C05458=1026.978,-87.134,412.335,166.934,44.993,158.253
C05459=1026.984,-86.885,412.325,166.937,44.991,158.253
C05460=1026.990,-86.635,412.315,166.940,44.988,158.253
C05461=1026.996,-86.385,412.304,166.943,44.986,158.253
C05462=1027.001,-86.135,412.294,166.946,44.984,158.253
C05463=1027.008,-85.886,412.284,166.948,44.981,158.252
C05464=1027.013,-85.636,412.274,166.952,44.979,158.252
C05465=1027.019,-85.386,412.264,166.954,44.976,158.252
C05466=1027.026,-85.103,412.252,166.958,44.974,158.252
C05467=1027.033,-84.819,412.240,166.961,44.971,158.252
C05468=1027.040,-84.534,412.228,166.965,44.968,158.252
C05469=1027.046,-84.250,412.217,166.968,44.966,158.252
C05470=1027.053,-84.001,412.207,166.971,44.964,158.251
C05471=1027.058,-83.751,412.196,166.974,44.961,158.251
C05472=1027.065,-83.502,412.186,166.977,44.959,158.251
C05473=1027.070,-83.252,412.176,166.980,44.956,158.251
C05474=1027.077,-83.002,412.165,166.983,44.954,158.251
C05475=1027.083,-82.752,412.155,166.986,44.952,158.251
C05476=1027.088,-82.502,412.144,166.989,44.949,158.251
C05477=1027.094,-82.252,412.135,166.992,44.947,158.251
C05478=1027.100,-82.003,412.124,166.995,44.944,158.250
C05479=1027.107,-81.754,412.114,166.997,44.942,158.250
C05480=1027.112,-81.503,412.103,167.001,44.939,158.250
C05481=1027.119,-81.254,412.093,167.003,44.937,158.250
C05482=1027.125,-81.003,412.083,167.007,44.934,158.250
C05483=1027.130,-80.754,412.072,167.009,44.932,158.250
C05484=1027.137,-80.505,412.061,167.013,44.929,158.250
C05485=1027.142,-80.255,412.051,167.015,44.927,158.250
C05486=1027.149,-80.006,412.041,167.019,44.925,158.250
C05487=1027.154,-79.756,412.030,167.021,44.922,158.249
C05488=1027.161,-79.505,412.020,167.024,44.920,158.249
C05489=1027.166,-79.256,412.009,167.027,44.918,158.249
C05490=1027.172,-79.006,411.998,167.030,44.916,158.249
C05491=1027.178,-78.757,411.988,167.032,44.914,158.249
C05492=1027.184,-78.507,411.977,167.036,44.911,158.249
C05493=1027.190,-78.257,411.966,167.038,44.909,158.249
C05494=1027.196,-78.007,411.955,167.042,44.907,158.249
C05495=1027.202,-77.758,411.944,167.044,44.905,158.248
C05496=1027.207,-77.508,411.934,167.047,44.903,158.248
C05497=1027.214,-77.258,411.924,167.050,44.900,158.248
C05498=1027.220,-77.008,411.913,167.053,44.898,158.248
C05499=1027.226,-76.759,411.902,167.056,44.896,158.248
C05500=1027.231,-76.509,411.891,167.059,44.893,158.248
C05501=1027.237,-76.260,411.880,167.062,44.891,158.248
C05502=1027.243,-76.010,411.869,167.065,44.889,158.248
C05503=1027.250,-75.760,411.859,167.068,44.887,158.248
C05504=1027.255,-75.510,411.848,167.070,44.884,158.247
C05505=1027.261,-75.261,411.838,167.074,44.882,158.247
C05506=1027.267,-75.011,411.827,167.076,44.880,158.247
C05507=1027.273,-74.761,411.815,167.079,44.877,158.247
C05508=1027.279,-74.512,411.805,167.082,44.875,158.247
C05509=1027.285,-74.262,411.794,167.085,44.873,158.247
C05510=1027.290,-74.013,411.783,167.089,44.871,158.247
C05511=1027.297,-73.763,411.772,167.091,44.868,158.247
C05512=1027.303,-73.513,411.761,167.094,44.866,158.247
C05513=1027.308,-73.264,411.750,167.096,44.864,158.246
C05514=1027.315,-73.013,411.739,167.100,44.862,158.246
C05515=1027.320,-72.764,411.728,167.102,44.860,158.246
C05516=1027.326,-72.514,411.717,167.105,44.858,158.246
C05517=1027.331,-72.265,411.705,167.109,44.856,158.246
C05518=1027.337,-72.014,411.694,167.111,44.854,158.246
C05519=1027.343,-71.765,411.683,167.113,44.851,158.246
C05520=1027.349,-71.515,411.672,167.117,44.849,158.246
C05521=1027.355,-71.265,411.661,167.120,44.847,158.246
C05522=1027.361,-71.016,411.650,167.122,44.845,158.246
C05523=1027.367,-70.766,411.639,167.125,44.843,158.246
C05524=1027.373,-70.517,411.627,167.129,44.841,158.246
C05525=1027.378,-70.267,411.616,167.131,44.839,158.245
C05526=1027.384,-70.017,411.605,167.134,44.837,158.245
C05527=1027.390,-69.767,411.594,167.137,44.834,158.245
C05528=1027.396,-69.518,411.583,167.140,44.832,158.245
C05529=1027.402,-69.268,411.572,167.142,44.830,158.245
C05530=1027.408,-68.987,411.559,167.146,44.828,158.245
C05531=1027.416,-68.704,411.546,167.149,44.825,158.245
C05532=1027.422,-68.423,411.534,167.152,44.823,158.245
C05533=1027.428,-68.141,411.521,167.155,44.820,158.245
C05534=1027.435,-67.891,411.509,167.158,44.818,158.244
C05535=1027.441,-67.641,411.498,167.161,44.816,158.244
C05536=1027.447,-67.391,411.487,167.164,44.814,158.244
C05537=1027.453,-67.142,411.476,167.167,44.812,158.244
C05538=1027.458,-66.892,411.465,167.170,44.810,158.244
C05539=1027.464,-66.642,411.453,167.173,44.807,158.244
C05540=1027.470,-66.393,411.442,167.175,44.805,158.244
C05541=1027.476,-66.143,411.430,167.178,44.803,158.244
C05542=1027.482,-65.894,411.419,167.181,44.801,158.244
C05543=1027.488,-65.644,411.408,167.184,44.799,158.244
C05544=1027.494,-65.394,411.396,167.187,44.797,158.244
C05545=1027.499,-65.144,411.385,167.190,44.794,158.243
C05546=1027.506,-64.895,411.373,167.193,44.792,158.243
C05547=1027.512,-64.645,411.362,167.195,44.790,158.243
C05548=1027.518,-64.395,411.351,167.199,44.788,158.243
C05549=1027.524,-64.146,411.340,167.201,44.786,158.243
C05550=1027.530,-63.896,411.328,167.204,44.784,158.243
C05551=1027.536,-63.646,411.317,167.206,44.781,158.243
C05552=1027.542,-63.397,411.305,167.210,44.779,158.243
C05553=1027.548,-63.147,411.294,167.213,44.777,158.243
C05554=1027.555,-62.898,411.282,167.215,44.775,158.242
C05555=1027.560,-62.648,411.271,167.219,44.773,158.242
C05556=1027.566,-62.398,411.259,167.221,44.770,158.242
C05557=1027.572,-62.149,411.248,167.224,44.768,158.242
C05558=1027.578,-61.899,411.237,167.227,44.766,158.242
C05559=1027.584,-61.650,411.225,167.230,44.764,158.242
C05560=1027.590,-61.399,411.213,167.233,44.762,158.242
C05561=1027.596,-61.150,411.202,167.235,44.760,158.242
C05562=1027.602,-60.900,411.190,167.239,44.757,158.242
C05563=1027.608,-60.651,411.179,167.241,44.755,158.241
C05564=1027.615,-60.401,411.167,167.244,44.753,158.241
C05565=1027.620,-60.151,411.156,167.247,44.751,158.241
C05566=1027.626,-59.902,411.144,167.250,44.749,158.241
C05567=1027.633,-59.652,411.133,167.252,44.747,158.241
C05568=1027.639,-59.403,411.121,167.255,44.745,158.241
C05569=1027.645,-59.152,411.110,167.259,44.742,158.241
C05570=1027.650,-58.903,411.098,167.261,44.740,158.241
C05571=1027.657,-58.653,411.086,167.264,44.738,158.241
C05572=1027.663,-58.404,411.075,167.267,44.736,158.240
C05573=1027.669,-58.154,411.064,167.270,44.734,158.240
C05574=1027.676,-57.904,411.052,167.272,44.732,158.240
C05575=1027.681,-57.655,411.040,167.276,44.729,158.240
C05576=1027.687,-57.405,411.028,167.278,44.727,158.240
C05577=1027.694,-57.155,411.017,167.281,44.725,158.240
C05578=1027.700,-56.906,411.005,167.284,44.723,158.240
C05579=1027.706,-56.656,410.993,167.287,44.721,158.240
C05580=1027.712,-56.407,410.982,167.289,44.718,158.240
C05581=1027.718,-56.157,410.970,167.292,44.716,158.239
C05582=1027.725,-55.907,410.959,167.296,44.714,158.239
C05583=1027.731,-55.658,410.947,167.298,44.712,158.239
C05584=1027.736,-55.408,410.935,167.301,44.709,158.239
C05585=1027.743,-55.158,410.923,167.303,44.707,158.239
C05586=1027.749,-54.909,410.912,167.307,44.705,158.239
C05587=1027.756,-54.660,410.900,167.309,44.703,158.239
C05588=1027.761,-54.409,410.888,167.312,44.700,158.239
C05589=1027.768,-54.159,410.876,167.315,44.698,158.239
C05590=1027.774,-53.911,410.864,167.318,44.696,158.238
C05591=1027.780,-53.660,410.853,167.321,44.694,158.238
C05592=1027.786,-53.410,410.841,167.324,44.692,158.238
C05593=1027.792,-53.162,410.829,167.327,44.690,158.238
C05594=1027.799,-52.881,410.816,167.329,44.687,158.238
C05595=1027.806,-52.600,410.802,167.333,44.685,158.238
C05596=1027.813,-52.319,410.790,167.336,44.682,158.238
C05597=1027.821,-52.038,410.776,167.340,44.680,158.238
C05598=1027.826,-51.788,410.764,167.342,44.678,158.237
C05599=1027.832,-51.539,410.753,167.345,44.675,158.237
C05600=1027.839,-51.290,410.741,167.347,44.673,158.237
C05601=1027.846,-51.040,410.729,167.351,44.671,158.237
C05602=1027.851,-50.789,410.717,167.353,44.668,158.237
C05603=1027.858,-50.540,410.705,167.356,44.666,158.237
C05604=1027.863,-50.291,410.693,167.358,44.664,158.237
C05605=1027.869,-50.041,410.680,167.362,44.662,158.237
C05606=1027.876,-49.791,410.668,167.365,44.660,158.236
C05607=1027.882,-49.541,410.656,167.367,44.658,158.236
C05608=1027.888,-49.293,410.644,167.370,44.656,158.236
C05609=1027.894,-49.043,410.631,167.372,44.654,158.236
C05610=1027.900,-48.793,410.619,167.376,44.652,158.236
C05611=1027.906,-48.543,410.607,167.379,44.650,158.236
C05612=1027.912,-48.294,410.595,167.381,44.648,158.236
C05613=1027.917,-48.044,410.582,167.384,44.646,158.236
C05614=1027.924,-47.795,410.570,167.386,44.644,158.236
C05615=1027.930,-47.545,410.558,167.389,44.642,158.236
C05616=1027.937,-47.295,410.546,167.393,44.640,158.236
C05617=1027.942,-47.046,410.534,167.395,44.638,158.235
C05618=1027.948,-46.796,410.521,167.398,44.636,158.235
C05619=1027.954,-46.546,410.509,167.400,44.634,158.235
C05620=1027.960,-46.297,410.497,167.403,44.632,158.235
C05621=1027.966,-46.047,410.484,167.407,44.630,158.235
C05622=1027.972,-45.798,410.472,167.409,44.628,158.235
C05623=1027.978,-45.548,410.460,167.412,44.626,158.235
C05624=1027.984,-45.298,410.447,167.414,44.624,158.235
C05625=1027.991,-45.048,410.435,167.417,44.622,158.235
C05626=1027.997,-44.799,410.423,167.420,44.619,158.235
C05627=1028.003,-44.549,410.410,167.423,44.617,158.234
C05628=1028.009,-44.300,410.399,167.426,44.615,158.234
C05629=1028.015,-44.050,410.386,167.428,44.614,158.234
C05630=1028.020,-43.800,410.373,167.431,44.612,158.234
C05631=1028.027,-43.551,410.361,167.433,44.610,158.234
C05632=1028.033,-43.301,410.348,167.437,44.607,158.234
C05633=1028.039,-43.051,410.336,167.440,44.605,158.234
C05634=1028.046,-42.802,410.324,167.442,44.604,158.234
C05635=1028.052,-42.552,410.311,167.445,44.602,158.234
C05636=1028.058,-42.302,410.299,167.447,44.600,158.234
C05637=1028.064,-42.052,410.287,167.451,44.597,158.233
C05638=1028.070,-41.804,410.274,167.453,44.595,158.233
C05639=1028.076,-41.554,410.261,167.456,44.593,158.233
C05640=1028.083,-41.304,410.249,167.459,44.591,158.233
C05641=1028.088,-41.055,410.237,167.461,44.589,158.233
C05642=1028.094,-40.805,410.224,167.464,44.587,158.233
C05643=1028.101,-40.556,410.211,167.467,44.585,158.233
C05644=1028.107,-40.306,410.199,167.470,44.583,158.233
C05645=1028.113,-40.056,410.186,167.473,44.581,158.233
C05646=1028.120,-39.806,410.174,167.475,44.579,158.232
C05647=1028.126,-39.557,410.161,167.478,44.576,158.232
C05648=1028.132,-39.307,410.149,167.481,44.574,158.232
C05649=1028.139,-39.058,410.137,167.484,44.572,158.232
C05650=1028.144,-38.808,410.124,167.486,44.570,158.232
C05651=1028.151,-38.558,410.111,167.489,44.568,158.232
C05652=1028.157,-38.309,410.098,167.492,44.566,158.232
C05653=1028.162,-38.059,410.086,167.494,44.564,158.232
C05654=1028.169,-37.809,410.072,167.497,44.562,158.232
C05655=1028.175,-37.560,410.060,167.499,44.560,158.231
C05656=1028.181,-37.310,410.047,167.503,44.558,158.231
C05657=1028.187,-37.060,410.034,167.506,44.557,158.231
C05658=1028.194,-36.780,410.019,167.508,44.554,158.231
C05659=1028.200,-36.500,410.006,167.512,44.552,158.231
C05660=1028.207,-36.220,409.991,167.514,44.550,158.231
C05661=1028.214,-35.940,409.977,167.518,44.548,158.231
C05662=1028.220,-35.690,409.963,167.521,44.546,158.231
C05663=1028.226,-35.440,409.951,167.523,44.544,158.231
C05664=1028.232,-35.191,409.938,167.526,44.542,158.231
C05665=1028.238,-34.941,409.925,167.528,44.540,158.231
C05666=1028.244,-34.691,409.913,167.531,44.538,158.230
C05667=1028.250,-34.442,409.899,167.534,44.536,158.230
C05668=1028.257,-34.193,409.887,167.536,44.534,158.230
C05669=1028.263,-33.943,409.874,167.539,44.532,158.230
C05670=1028.269,-33.693,409.861,167.542,44.530,158.230
C05671=1028.276,-33.443,409.848,167.545,44.528,158.230
C05672=1028.282,-33.194,409.835,167.548,44.526,158.230
C05673=1028.288,-32.944,409.822,167.550,44.524,158.230
C05674=1028.294,-32.695,409.809,167.553,44.522,158.230
C05675=1028.300,-32.445,409.796,167.555,44.520,158.230
C05676=1028.306,-32.196,409.783,167.558,44.519,158.229
C05677=1028.312,-31.946,409.770,167.561,44.517,158.229
C05678=1028.318,-31.697,409.757,167.563,44.515,158.229
C05679=1028.324,-31.447,409.745,167.567,44.512,158.229
C05680=1028.330,-31.198,409.731,167.570,44.511,158.229
C05681=1028.337,-30.948,409.718,167.572,44.509,158.229
C05682=1028.343,-30.698,409.705,167.575,44.507,158.229
C05683=1028.349,-30.448,409.692,167.577,44.505,158.229
C05684=1028.356,-30.199,409.679,167.580,44.502,158.228
C05685=1028.361,-29.949,409.666,167.582,44.500,158.228
C05686=1028.368,-29.700,409.653,167.585,44.498,158.228
C05687=1028.374,-29.450,409.640,167.587,44.496,158.228
C05688=1028.380,-29.201,409.627,167.591,44.494,158.228
C05689=1028.387,-28.951,409.613,167.594,44.492,158.228
C05690=1028.393,-28.701,409.601,167.596,44.490,158.228
C05691=1028.399,-28.452,409.587,167.599,44.488,158.228
C05692=1028.405,-28.203,409.574,167.602,44.486,158.228
C05693=1028.411,-27.953,409.562,167.604,44.484,158.228
C05694=1028.418,-27.703,409.548,167.607,44.482,158.227
C05695=1028.424,-27.453,409.535,167.609,44.480,158.227
C05696=1028.430,-27.204,409.521,167.612,44.478,158.227
C05697=1028.436,-26.954,409.509,167.615,44.476,158.227
C05698=1028.442,-26.705,409.496,167.617,44.475,158.227
C05699=1028.448,-26.456,409.482,167.620,44.473,158.227
C05700=1028.455,-26.205,409.468,167.623,44.470,158.227
C05701=1028.461,-25.956,409.455,167.626,44.468,158.227
C05702=1028.467,-25.707,409.442,167.629,44.467,158.227
C05703=1028.473,-25.457,409.429,167.631,44.465,158.227
C05704=1028.478,-25.207,409.415,167.634,44.463,158.227
C05705=1028.485,-24.958,409.402,167.637,44.461,158.226
C05706=1028.491,-24.708,409.388,167.639,44.459,158.226
C05707=1028.498,-24.459,409.375,167.642,44.457,158.226
C05708=1028.503,-24.209,409.361,167.644,44.456,158.226
C05709=1028.509,-23.960,409.348,167.647,44.454,158.226
C05710=1028.516,-23.710,409.334,167.650,44.452,158.226
C05711=1028.522,-23.460,409.322,167.652,44.450,158.226
C05712=1028.527,-23.211,409.308,167.655,44.448,158.226
C05713=1028.534,-22.961,409.295,167.657,44.446,158.226
C05714=1028.540,-22.718,409.281,167.660,44.445,158.226
C05715=1028.546,-22.474,409.268,167.663,44.443,158.226
C05716=1028.552,-22.230,409.255,167.665,44.441,158.225
C05717=1028.558,-21.987,409.241,167.668,44.439,158.225
C05718=1028.564,-21.743,409.228,167.671,44.437,158.225
C05719=1028.570,-21.499,409.215,167.673,44.435,158.225
C05720=1028.576,-21.255,409.201,167.676,44.433,158.225
C05721=1028.582,-21.011,409.189,167.678,44.431,158.225
C05722=1028.590,-20.718,409.173,167.681,44.429,158.225
C05723=1028.597,-20.426,409.157,167.685,44.427,158.225
C05724=1028.605,-20.133,409.141,167.687,44.424,158.224
C05725=1028.611,-19.841,409.125,167.691,44.422,158.224
C05726=1028.618,-19.591,409.111,167.693,44.420,158.224
C05727=1028.624,-19.341,409.098,167.696,44.418,158.224
C05728=1028.630,-19.092,409.084,167.698,44.416,158.224
C05729=1028.637,-18.842,409.070,167.701,44.414,158.224
C05730=1028.643,-18.593,409.057,167.704,44.412,158.224
C05731=1028.648,-18.343,409.043,167.706,44.410,158.224
C05732=1028.655,-18.093,409.030,167.709,44.408,158.224
C05733=1028.661,-17.844,409.016,167.711,44.406,158.223
C05734=1028.668,-17.594,409.003,167.714,44.405,158.223
C05735=1028.674,-17.344,408.989,167.717,44.403,158.223
C05736=1028.680,-17.095,408.976,167.719,44.401,158.223
C05737=1028.686,-16.846,408.962,167.722,44.399,158.223
C05738=1028.692,-16.596,408.947,167.724,44.397,158.223
C05739=1028.699,-16.347,408.934,167.727,44.395,158.223
C05740=1028.705,-16.097,408.920,167.730,44.393,158.223
C05741=1028.711,-15.847,408.907,167.732,44.391,158.223
C05742=1028.717,-15.598,408.893,167.735,44.389,158.222
C05743=1028.724,-15.348,408.880,167.737,44.387,158.222
C05744=1028.730,-15.099,408.865,167.740,44.385,158.222
C05745=1028.737,-14.849,408.851,167.743,44.384,158.222
C05746=1028.742,-14.599,408.838,167.746,44.382,158.222
C05747=1028.747,-14.350,408.824,167.748,44.380,158.222
C05748=1028.755,-14.101,408.809,167.751,44.378,158.222
C05749=1028.760,-13.851,408.796,167.753,44.376,158.222
C05750=1028.767,-13.601,408.782,167.756,44.374,158.222
C05751=1028.772,-13.351,408.768,167.759,44.372,158.222
C05752=1028.779,-13.103,408.754,167.761,44.370,158.221
C05753=1028.785,-12.853,408.740,167.764,44.369,158.222
C05754=1028.791,-12.603,408.727,167.767,44.367,158.221
C05755=1028.798,-12.354,408.712,167.769,44.365,158.221
C05756=1028.803,-12.104,408.698,167.772,44.363,158.221
C05757=1028.810,-11.854,408.684,167.774,44.361,158.221
C05758=1028.816,-11.605,408.670,167.777,44.359,158.221
C05759=1028.822,-11.356,408.656,167.780,44.357,158.221
C05760=1028.828,-11.106,408.641,167.782,44.355,158.221
C05761=1028.834,-10.857,408.628,167.785,44.353,158.221
C05762=1028.841,-10.607,408.614,167.788,44.352,158.221
C05763=1028.847,-10.358,408.600,167.790,44.350,158.221
C05764=1028.853,-10.108,408.586,167.793,44.348,158.220
C05765=1028.859,-9.858,408.572,167.795,44.346,158.220
C05766=1028.866,-9.609,408.557,167.798,44.344,158.220
C05767=1028.871,-9.359,408.544,167.801,44.343,158.220
C05768=1028.878,-9.110,408.529,167.803,44.341,158.220
C05769=1028.884,-8.860,408.515,167.806,44.339,158.220
C05770=1028.891,-8.611,408.501,167.808,44.337,158.220
C05771=1028.896,-8.361,408.487,167.811,44.335,158.220
C05772=1028.903,-8.112,408.472,167.813,44.333,158.219
C05773=1028.909,-7.862,408.459,167.815,44.331,158.219
C05774=1028.915,-7.612,408.445,167.818,44.329,158.219
C05775=1028.922,-7.364,408.431,167.821,44.328,158.219
C05776=1028.928,-7.113,408.416,167.823,44.326,158.219
C05777=1028.933,-6.864,408.402,167.826,44.324,158.219
C05778=1028.940,-6.614,408.388,167.828,44.322,158.219
C05779=1028.947,-6.365,408.373,167.831,44.320,158.219
C05780=1028.953,-6.115,408.360,167.834,44.318,158.219
C05781=1028.959,-5.866,408.345,167.836,44.316,158.219
C05782=1028.965,-5.616,408.331,167.839,44.314,158.218
C05783=1028.972,-5.367,408.317,167.841,44.312,158.218
C05784=1028.978,-5.118,408.302,167.844,44.310,158.218
C05785=1028.984,-4.868,408.289,167.847,44.309,158.218
C05786=1028.991,-4.585,408.273,167.849,44.307,158.218
C05787=1028.998,-4.302,408.256,167.853,44.304,158.218
C05788=1029.006,-4.020,408.240,167.855,44.302,158.218
C05789=1029.013,-3.736,408.224,167.858,44.300,158.218
C05790=1029.018,-3.487,408.209,167.861,44.298,158.217
C05791=1029.025,-3.238,408.194,167.863,44.297,158.217
C05792=1029.031,-2.988,408.179,167.866,44.295,158.217
C05793=1029.037,-2.739,408.165,167.869,44.293,158.217
C05794=1029.043,-2.489,408.151,167.871,44.291,158.217
C05795=1029.049,-2.240,408.136,167.874,44.289,158.217
C05796=1029.056,-1.991,408.122,167.877,44.288,158.217
C05797=1029.061,-1.741,408.108,167.878,44.286,158.217
C05798=1029.068,-1.491,408.093,167.881,44.284,158.217
C05799=1029.074,-1.242,408.078,167.883,44.282,158.217
C05800=1029.080,-0.993,408.063,167.886,44.281,158.217
C05801=1029.086,-0.742,408.049,167.889,44.279,158.216
C05802=1029.092,-0.494,408.034,167.891,44.277,158.216
C05803=1029.098,-0.244,408.020,167.894,44.275,158.216
C05804=1029.105,0.006,408.005,167.897,44.273,158.216
C05805=1029.110,0.255,407.990,167.898,44.271,158.216
C05806=1029.116,0.505,407.976,167.901,44.270,158.216
C05807=1029.123,0.755,407.961,167.904,44.268,158.216
C05808=1029.129,1.004,407.946,167.906,44.266,158.216
C05809=1029.135,1.253,407.931,167.909,44.264,158.216
C05810=1029.141,1.503,407.916,167.911,44.262,158.216
C05811=1029.147,1.752,407.902,167.914,44.261,158.216
C05812=1029.153,2.002,407.888,167.917,44.259,158.215
C05813=1029.160,2.252,407.873,167.918,44.258,158.215
C05814=1029.166,2.500,407.859,167.921,44.256,158.215
C05815=1029.173,2.750,407.844,167.924,44.254,158.215
C05816=1029.179,3.000,407.829,167.926,44.252,158.215
C05817=1029.185,3.249,407.814,167.929,44.251,158.215
C05818=1029.191,3.498,407.799,167.932,44.249,158.215
C05819=1029.197,3.748,407.784,167.934,44.247,158.215
C05820=1029.203,3.997,407.770,167.937,44.245,158.215
C05821=1029.210,4.247,407.755,167.939,44.243,158.214
C05822=1029.216,4.496,407.740,167.941,44.241,158.214
C05823=1029.221,4.746,407.726,167.944,44.239,158.214
C05824=1029.228,4.996,407.711,167.947,44.238,158.214
C05825=1029.234,5.245,407.696,167.949,44.236,158.214
C05826=1029.241,5.495,407.681,167.952,44.234,158.214
C05827=1029.246,5.744,407.666,167.954,44.232,158.214
C05828=1029.253,5.993,407.652,167.957,44.230,158.214
C05829=1029.259,6.243,407.637,167.960,44.228,158.214
C05830=1029.266,6.493,407.622,167.961,44.227,158.213
C05831=1029.271,6.742,407.607,167.964,44.225,158.213
C05832=1029.278,6.991,407.592,167.966,44.223,158.213
C05833=1029.284,7.241,407.577,167.969,44.221,158.213
C05834=1029.290,7.491,407.562,167.972,44.220,158.213
C05835=1029.297,7.740,407.547,167.974,44.218,158.213
C05836=1029.303,7.989,407.533,167.977,44.216,158.213
C05837=1029.309,8.239,407.518,167.980,44.214,158.213
C05838=1029.315,8.489,407.503,167.981,44.212,158.213
C05839=1029.322,8.738,407.487,167.984,44.210,158.212
C05840=1029.328,8.987,407.472,167.986,44.208,158.212
C05841=1029.334,9.236,407.458,167.989,44.206,158.212
C05842=1029.341,9.486,407.443,167.992,44.204,158.212
C05843=1029.347,9.736,407.428,167.994,44.202,158.212
C05844=1029.353,9.985,407.413,167.997,44.200,158.212
C05845=1029.360,10.235,407.398,167.999,44.199,158.212
C05846=1029.366,10.484,407.383,168.002,44.197,158.212
C05847=1029.372,10.734,407.368,168.004,44.196,158.212
C05848=1029.378,10.983,407.353,168.006,44.194,158.211
C05849=1029.385,11.232,407.338,168.009,44.192,158.211
C05850=1029.392,11.517,407.321,168.011,44.189,158.211
C05851=1029.399,11.802,407.304,168.015,44.187,158.211
C05852=1029.407,12.087,407.287,168.018,44.185,158.211
C05853=1029.414,12.371,407.269,168.020,44.183,158.211
C05854=1029.420,12.621,407.254,168.023,44.181,158.211
C05855=1029.427,12.871,407.240,168.025,44.179,158.210
C05856=1029.433,13.120,407.225,168.028,44.177,158.210
C05857=1029.440,13.369,407.209,168.031,44.175,158.210
C05858=1029.445,13.618,407.194,168.033,44.174,158.210
C05859=1029.452,13.868,407.179,168.036,44.172,158.210
C05860=1029.458,14.118,407.164,168.037,44.170,158.210
C05861=1029.464,14.367,407.148,168.040,44.168,158.210
C05862=1029.471,14.617,407.133,168.043,44.166,158.210
C05863=1029.477,14.866,407.118,168.046,44.165,158.210
C05864=1029.484,15.115,407.103,168.048,44.163,158.209
C05865=1029.489,15.365,407.087,168.051,44.161,158.209
C05866=1029.496,15.615,407.072,168.052,44.159,158.209
C05867=1029.502,15.863,407.057,168.055,44.157,158.209
C05868=1029.508,16.113,407.042,168.058,44.155,158.209
C05869=1029.514,16.363,407.026,168.060,44.154,158.209
C05870=1029.520,16.612,407.011,168.063,44.152,158.209
C05871=1029.527,16.862,406.996,168.065,44.151,158.209
C05872=1029.532,17.112,406.980,168.067,44.149,158.209
C05873=1029.539,17.361,406.965,168.070,44.147,158.208
C05874=1029.546,17.610,406.950,168.072,44.145,158.208
C05875=1029.552,17.859,406.934,168.075,44.143,158.208
C05876=1029.558,18.109,406.918,168.078,44.142,158.208
C05877=1029.564,18.359,406.903,168.079,44.140,158.208
C05878=1029.571,18.608,406.888,168.082,44.138,158.208
C05879=1029.577,18.858,406.872,168.085,44.136,158.208
C05880=1029.583,19.107,406.857,168.087,44.134,158.208
C05881=1029.589,19.356,406.842,168.090,44.132,158.208
C05882=1029.596,19.605,406.826,168.091,44.130,158.207
C05883=1029.601,19.855,406.811,168.094,44.129,158.207
C05884=1029.608,20.104,406.795,168.097,44.127,158.207
C05885=1029.614,20.354,406.780,168.099,44.125,158.207
C05886=1029.620,20.603,406.764,168.102,44.123,158.207
C05887=1029.626,20.853,406.748,168.104,44.122,158.207
C05888=1029.633,21.102,406.733,168.106,44.121,158.207
C05889=1029.639,21.352,406.718,168.109,44.119,158.207
C05890=1029.645,21.601,406.702,168.112,44.117,158.207
C05891=1029.651,21.851,406.687,168.114,44.115,158.206
C05892=1029.657,22.100,406.670,168.116,44.113,158.206
C05893=1029.664,22.350,406.655,168.119,44.111,158.206
C05894=1029.670,22.599,406.639,168.121,44.110,158.206
C05895=1029.676,22.848,406.623,168.124,44.108,158.206
C05896=1029.682,23.098,406.608,168.127,44.106,158.206
C05897=1029.689,23.347,406.592,168.128,44.104,158.206
C05898=1029.695,23.597,406.577,168.131,44.102,158.206
C05899=1029.701,23.846,406.561,168.133,44.100,158.206
C05900=1029.708,24.095,406.545,168.136,44.099,158.206
C05901=1029.713,24.345,406.530,168.139,44.097,158.205
C05902=1029.720,24.594,406.514,168.140,44.096,158.205
C05903=1029.726,24.843,406.498,168.143,44.094,158.205
C05904=1029.732,25.093,406.483,168.146,44.092,158.205
C05905=1029.739,25.343,406.466,168.148,44.090,158.205
C05906=1029.746,25.592,406.451,168.151,44.088,158.205
C05907=1029.752,25.842,406.436,168.152,44.086,158.205
C05908=1029.758,26.091,406.420,168.155,44.085,158.205
C05909=1029.765,26.340,406.404,168.158,44.083,158.204
C05910=1029.770,26.590,406.388,168.160,44.081,158.204
C05911=1029.777,26.839,406.373,168.162,44.079,158.204
C05912=1029.783,27.089,406.356,168.165,44.078,158.204
C05913=1029.789,27.338,406.340,168.167,44.076,158.204
C05914=1029.797,27.624,406.323,168.170,44.074,158.204
C05915=1029.804,27.910,406.305,168.172,44.072,158.204
C05916=1029.811,28.196,406.286,168.176,44.070,158.204
C05917=1029.818,28.482,406.268,168.179,44.068,158.203
C05918=1029.823,28.732,406.252,168.181,44.066,158.203
C05919=1029.830,28.981,406.236,168.183,44.064,158.203
C05920=1029.836,29.230,406.220,168.186,44.063,158.203
C05921=1029.842,29.479,406.204,168.188,44.061,158.203
C05922=1029.849,29.729,406.188,168.191,44.059,158.203
C05923=1029.855,29.979,406.172,168.193,44.057,158.203
C05924=1029.861,30.228,406.155,168.195,44.056,158.203
C05925=1029.868,30.478,406.140,168.198,44.054,158.203
C05926=1029.874,30.727,406.124,168.201,44.052,158.202
C05927=1029.879,30.976,406.108,168.202,44.051,158.202
C05928=1029.886,31.225,406.092,168.205,44.049,158.202
C05929=1029.892,31.475,406.076,168.208,44.047,158.202
C05930=1029.899,31.725,406.059,168.210,44.046,158.202
C05931=1029.905,31.974,406.044,168.212,44.044,158.202
C05932=1029.911,32.223,406.027,168.214,44.042,158.202
C05933=1029.917,32.472,406.011,168.217,44.040,158.202
C05934=1029.923,32.722,405.995,168.220,44.039,158.202
C05935=1029.930,32.971,405.979,168.221,44.037,158.201
C05936=1029.936,33.221,405.964,168.224,44.035,158.201
C05937=1029.942,33.471,405.947,168.227,44.033,158.201
C05938=1029.949,33.720,405.931,168.229,44.031,158.201
C05939=1029.955,33.969,405.915,168.231,44.030,158.201
C05940=1029.961,34.219,405.899,168.234,44.028,158.201
C05941=1029.967,34.468,405.883,168.236,44.026,158.201
C05942=1029.973,34.717,405.867,168.239,44.025,158.201
C05943=1029.980,34.967,405.850,168.240,44.023,158.201
C05944=1029.986,35.216,405.834,168.243,44.021,158.200
C05945=1029.993,35.465,405.818,168.246,44.019,158.200
C05946=1029.998,35.715,405.802,168.248,44.017,158.200
C05947=1030.005,35.965,405.786,168.250,44.016,158.200
C05948=1030.012,36.214,405.770,168.253,44.014,158.200
C05949=1030.018,36.463,405.754,168.255,44.012,158.200
C05950=1030.024,36.712,405.737,168.258,44.010,158.200
C05951=1030.030,36.961,405.720,168.260,44.009,158.200
C05952=1030.037,37.211,405.704,168.262,44.007,158.199
C05953=1030.043,37.460,405.688,168.265,44.006,158.199
C05954=1030.049,37.710,405.672,168.268,44.004,158.199
C05955=1030.055,37.959,405.656,168.269,44.002,158.199
C05956=1030.062,38.209,405.639,168.272,44.000,158.199
C05957=1030.068,38.458,405.623,168.275,43.999,158.199
C05958=1030.074,38.707,405.606,168.276,43.997,158.199
C05959=1030.080,38.956,405.590,168.279,43.995,158.199
C05960=1030.086,39.206,405.573,168.281,43.993,158.199
C05961=1030.092,39.456,405.557,168.284,43.992,158.199
C05962=1030.098,39.705,405.540,168.286,43.990,158.198
C05963=1030.104,39.955,405.524,168.288,43.988,158.198
C05964=1030.110,40.203,405.507,168.291,43.986,158.198
C05965=1030.117,40.453,405.491,168.294,43.985,158.198
C05966=1030.123,40.703,405.474,168.295,43.984,158.198
C05967=1030.129,40.952,405.458,168.298,43.982,158.198
C05968=1030.135,41.201,405.441,168.301,43.980,158.198
C05969=1030.142,41.451,405.424,168.302,43.978,158.198
C05970=1030.148,41.700,405.408,168.305,43.977,158.198
C05971=1030.154,41.950,405.392,168.308,43.975,158.197
C05972=1030.161,42.199,405.375,168.310,43.973,158.197
C05973=1030.167,42.448,405.359,168.312,43.971,158.197
C05974=1030.173,42.697,405.343,168.315,43.969,158.197
C05975=1030.179,42.946,405.326,168.317,43.968,158.197
C05976=1030.185,43.196,405.308,168.319,43.966,158.197
C05977=1030.191,43.446,405.292,168.322,43.965,158.197
C05978=1030.199,43.731,405.273,168.324,43.963,158.197
C05979=1030.205,44.018,405.254,168.327,43.961,158.197
C05980=1030.212,44.303,405.234,168.330,43.959,158.196
C05981=1030.219,44.589,405.215,168.332,43.958,158.196
C05982=1030.225,44.838,405.198,168.335,43.956,158.196
C05983=1030.231,45.089,405.181,168.337,43.954,158.196
C05984=1030.237,45.338,405.165,168.339,43.953,158.196
C05985=1030.243,45.587,405.148,168.342,43.951,158.196
C05986=1030.250,45.837,405.131,168.344,43.949,158.196
C05987=1030.256,46.086,405.114,168.346,43.948,158.196
C05988=1030.262,46.335,405.098,168.349,43.946,158.196
C05989=1030.268,46.584,405.080,168.352,43.944,158.195
C05990=1030.274,46.834,405.064,168.353,43.943,158.195
C05991=1030.281,47.083,405.047,168.356,43.941,158.195
C05992=1030.286,47.333,405.030,168.359,43.939,158.195
C05993=1030.293,47.582,405.013,168.360,43.938,158.195
C05994=1030.299,47.831,404.997,168.363,43.936,158.195
C05995=1030.305,48.080,404.979,168.366,43.934,158.195
C05996=1030.311,48.330,404.962,168.367,43.933,158.195
C05997=1030.317,48.579,404.945,168.370,43.931,158.195
C05998=1030.323,48.829,404.929,168.373,43.930,158.195
C05999=1030.330,49.078,404.912,168.374,43.928,158.194
C06000=1030.335,49.327,404.895,168.377,43.927,158.194
C06001=1030.342,49.577,404.878,168.380,43.925,158.194
C06002=1030.348,49.826,404.861,168.381,43.923,158.194
C06003=1030.355,50.075,404.844,168.384,43.922,158.194
C06004=1030.360,50.324,404.826,168.387,43.920,158.194
C06005=1030.366,50.574,404.810,168.389,43.918,158.194
C06006=1030.373,50.823,404.793,168.391,43.916,158.194
C06007=1030.379,51.073,404.777,168.394,43.915,158.194
C06008=1030.385,51.322,404.759,168.396,43.913,158.194
C06009=1030.391,51.571,404.742,168.398,43.911,158.193
C06010=1030.397,51.820,404.725,168.401,43.910,158.193
C06011=1030.404,52.070,404.708,168.403,43.908,158.193
C06012=1030.409,52.320,404.691,168.405,43.907,158.193
C06013=1030.416,52.569,404.674,168.408,43.905,158.193
C06014=1030.422,52.818,404.657,168.410,43.903,158.193
C06015=1030.429,53.068,404.640,168.412,43.902,158.193
C06016=1030.434,53.317,404.623,168.415,43.900,158.193
C06017=1030.441,53.565,404.606,168.417,43.898,158.192
C06018=1030.447,53.816,404.589,168.420,43.896,158.192
C06019=1030.453,54.065,404.572,168.421,43.894,158.192
C06020=1030.460,54.314,404.554,168.424,43.893,158.192
C06021=1030.466,54.563,404.538,168.427,43.891,158.192
C06022=1030.472,54.813,404.521,168.428,43.890,158.192
C06023=1030.478,55.062,404.503,168.431,43.888,158.192
C06024=1030.485,55.311,404.486,168.434,43.886,158.192
C06025=1030.491,55.561,404.469,168.435,43.885,158.192
C06026=1030.498,55.810,404.452,168.438,43.883,158.191
C06027=1030.503,56.059,404.435,168.441,43.881,158.191
C06028=1030.510,56.309,404.418,168.443,43.879,158.191
C06029=1030.516,56.558,404.401,168.445,43.877,158.191
C06030=1030.522,56.808,404.383,168.448,43.876,158.191
C06031=1030.528,57.056,404.366,168.450,43.874,158.191
C06032=1030.535,57.306,404.349,168.452,43.873,158.191
C06033=1030.541,57.555,404.332,168.455,43.871,158.190
C06034=1030.547,57.805,404.315,168.457,43.869,158.190
C06035=1030.554,58.054,404.298,168.460,43.868,158.190
C06036=1030.560,58.303,404.280,168.462,43.866,158.190
C06037=1030.566,58.553,404.263,168.464,43.864,158.190
C06038=1030.572,58.802,404.246,168.467,43.862,158.190
C06039=1030.579,59.052,404.229,168.468,43.860,158.190
C06040=1030.586,59.300,404.212,168.471,43.858,158.190
C06041=1030.592,59.550,404.194,168.474,43.857,158.189
C06042=1030.599,59.836,404.174,168.476,43.855,158.189
C06043=1030.606,60.122,404.154,168.479,43.853,158.189
C06044=1030.613,60.406,404.135,168.481,43.851,158.189
C06045=1030.620,60.692,404.116,168.484,43.849,158.189
C06046=1030.627,60.942,404.098,168.487,43.847,158.189
C06047=1030.633,61.192,404.080,168.489,43.845,158.189
C06048=1030.640,61.440,404.063,168.491,43.844,158.188
C06049=1030.647,61.690,404.046,168.493,43.842,158.188
C06050=1030.652,61.939,404.028,168.496,43.840,158.188
C06051=1030.659,62.189,404.012,168.499,43.839,158.188
C06052=1030.665,62.438,403.994,168.500,43.837,158.188
C06053=1030.672,62.687,403.977,168.503,43.835,158.188
C06054=1030.678,62.937,403.960,168.506,43.833,158.188
C06055=1030.684,63.185,403.943,168.508,43.831,158.188
C06056=1030.691,63.435,403.925,168.510,43.830,158.187
C06057=1030.697,63.685,403.907,168.513,43.828,158.187
C06058=1030.703,63.934,403.890,168.515,43.826,158.187
C06059=1030.709,64.183,403.872,168.517,43.825,158.187
C06060=1030.716,64.433,403.854,168.520,43.823,158.187
C06061=1030.722,64.682,403.837,168.522,43.822,158.187
C06062=1030.728,64.931,403.820,168.524,43.820,158.187
C06063=1030.734,65.180,403.803,168.527,43.818,158.187
C06064=1030.740,65.430,403.785,168.529,43.816,158.187
C06065=1030.746,65.679,403.767,168.531,43.815,158.187
C06066=1030.753,65.928,403.749,168.534,43.813,158.186
C06067=1030.759,66.177,403.731,168.536,43.811,158.186
C06068=1030.766,66.427,403.714,168.538,43.810,158.186
C06069=1030.772,66.676,403.696,168.541,43.808,158.186
C06070=1030.778,66.926,403.678,168.543,43.807,158.186
C06071=1030.784,67.174,403.661,168.545,43.805,158.186
C06072=1030.790,67.424,403.643,168.548,43.803,158.186
C06073=1030.796,67.674,403.625,168.550,43.802,158.186
C06074=1030.803,67.922,403.608,168.553,43.800,158.185
C06075=1030.809,68.172,403.590,168.555,43.798,158.185
C06076=1030.815,68.421,403.572,168.557,43.796,158.185
C06077=1030.821,68.670,403.555,168.560,43.795,158.185
C06078=1030.827,68.920,403.537,168.562,43.793,158.185
C06079=1030.834,69.169,403.518,168.564,43.791,158.185
C06080=1030.839,69.418,403.501,168.567,43.790,158.185
C06081=1030.846,69.667,403.483,168.569,43.789,158.185
C06082=1030.852,69.917,403.465,168.571,43.787,158.185
C06083=1030.858,70.166,403.448,168.574,43.785,158.184
C06084=1030.864,70.415,403.429,168.576,43.784,158.184
C06085=1030.871,70.665,403.412,168.578,43.782,158.184
C06086=1030.877,70.914,403.394,168.581,43.780,158.184
C06087=1030.883,71.163,403.376,168.583,43.779,158.184
C06088=1030.889,71.413,403.358,168.585,43.777,158.184
C06089=1030.895,71.662,403.340,168.587,43.775,158.184
C06090=1030.901,71.911,403.323,168.590,43.774,158.184
C06091=1030.908,72.160,403.304,168.592,43.772,158.184
C06092=1030.914,72.410,403.286,168.594,43.771,158.183
C06093=1030.920,72.659,403.269,168.597,43.769,158.183
C06094=1030.926,72.908,403.250,168.599,43.767,158.183
C06095=1030.932,73.158,403.232,168.601,43.766,158.183
C06096=1030.939,73.407,403.214,168.604,43.764,158.183
C06097=1030.945,73.656,403.196,168.606,43.763,158.183
C06098=1030.951,73.905,403.179,168.608,43.761,158.183
C06099=1030.957,74.155,403.160,168.611,43.759,158.183
C06100=1030.963,74.404,403.142,168.613,43.757,158.182
C06101=1030.969,74.653,403.124,168.616,43.756,158.182
C06102=1030.976,74.902,403.106,168.618,43.754,158.182
C06103=1030.982,75.152,403.088,168.620,43.752,158.182
C06104=1030.989,75.401,403.070,168.623,43.751,158.182
C06105=1030.994,75.650,403.052,168.625,43.749,158.182
C06106=1031.001,75.935,403.032,168.627,43.748,158.182
C06107=1031.009,76.221,403.011,168.630,43.746,158.182
C06108=1031.016,76.506,402.990,168.633,43.744,158.182
C06109=1031.023,76.792,402.969,168.635,43.742,158.181
C06110=1031.029,77.041,402.951,168.638,43.740,158.181
C06111=1031.035,77.290,402.932,168.640,43.738,158.181
C06112=1031.042,77.540,402.915,168.642,43.737,158.181
C06113=1031.048,77.789,402.896,168.645,43.735,158.181
C06114=1031.054,78.038,402.879,168.647,43.733,158.181
C06115=1031.060,78.288,402.860,168.649,43.732,158.181
C06116=1031.066,78.537,402.842,168.652,43.731,158.181
C06117=1031.072,78.786,402.823,168.655,43.729,158.181
C06118=1031.078,79.036,402.805,168.656,43.728,158.180
C06119=1031.084,79.285,402.787,168.659,43.726,158.180
C06120=1031.091,79.534,402.768,168.662,43.725,158.180
C06121=1031.097,79.783,402.750,168.663,43.723,158.180
C06122=1031.103,80.033,402.732,168.666,43.721,158.180
C06123=1031.109,80.282,402.714,168.669,43.720,158.180
C06124=1031.115,80.531,402.695,168.670,43.718,158.180
C06125=1031.121,80.780,402.676,168.673,43.717,158.180
C06126=1031.127,81.030,402.658,168.676,43.715,158.180
C06127=1031.133,81.279,402.639,168.677,43.713,158.180
C06128=1031.140,81.528,402.621,168.680,43.712,158.180
C06129=1031.145,81.777,402.603,168.682,43.710,158.179
C06130=1031.152,82.026,402.585,168.684,43.708,158.179
C06131=1031.158,82.275,402.566,168.687,43.707,158.179
C06132=1031.164,82.525,402.548,168.689,43.706,158.179
C06133=1031.170,82.775,402.529,168.691,43.704,158.179
C06134=1031.176,83.024,402.510,168.694,43.703,158.179
C06135=1031.182,83.273,402.492,168.696,43.701,158.179
C06136=1031.188,83.522,402.474,168.699,43.699,158.179
C06137=1031.195,83.771,402.455,168.701,43.698,158.179
C06138=1031.201,84.020,402.437,168.703,43.696,158.178
C06139=1031.207,84.270,402.419,168.706,43.694,158.178
C06140=1031.214,84.519,402.400,168.708,43.693,158.178
C06141=1031.219,84.768,402.381,168.710,43.691,158.178
C06142=1031.226,85.018,402.362,168.713,43.689,158.178
C06143=1031.232,85.267,402.344,168.715,43.688,158.178
C06144=1031.238,85.516,402.326,168.717,43.686,158.178
C06145=1031.244,85.765,402.307,168.720,43.685,158.178
C06146=1031.251,86.014,402.289,168.722,43.683,158.178
C06147=1031.257,86.264,402.271,168.724,43.682,158.177
C06148=1031.263,86.513,402.252,168.727,43.680,158.177
C06149=1031.269,86.762,402.233,168.729,43.678,158.177
C06150=1031.275,87.011,402.214,168.732,43.677,158.177
C06151=1031.282,87.260,402.196,168.734,43.675,158.177
C06152=1031.288,87.510,402.177,168.736,43.673,158.177
C06153=1031.294,87.759,402.159,168.739,43.672,158.177
C06154=1031.301,88.008,402.140,168.741,43.670,158.177
C06155=1031.307,88.258,402.122,168.743,43.668,158.176
C06156=1031.313,88.507,402.102,168.746,43.667,158.176
C06157=1031.319,88.756,402.084,168.748,43.666,158.176
C06158=1031.325,89.005,402.065,168.750,43.664,158.176
C06159=1031.331,89.254,402.048,168.753,43.662,158.176
C06160=1031.337,89.503,402.029,168.755,43.661,158.176
C06161=1031.344,89.753,402.010,168.757,43.659,158.176
C06162=1031.350,90.002,401.991,168.760,43.657,158.176
C06163=1031.356,90.251,401.972,168.762,43.656,158.176
C06164=1031.362,90.501,401.953,168.765,43.654,158.175
C06165=1031.368,90.750,401.934,168.767,43.652,158.175
C06166=1031.374,90.999,401.915,168.769,43.651,158.175
C06167=1031.380,91.248,401.897,168.772,43.649,158.175
C06168=1031.387,91.497,401.878,168.774,43.648,158.175
C06169=1031.392,91.747,401.859,168.776,43.646,158.175
C06170=1031.399,92.032,401.837,168.779,43.645,158.175
C06171=1031.406,92.318,401.815,168.781,43.643,158.175
C06172=1031.414,92.603,401.794,168.784,43.642,158.175
C06173=1031.421,92.888,401.772,168.788,43.639,158.175
C06174=1031.426,93.137,401.752,168.789,43.638,158.174
C06175=1031.433,93.386,401.734,168.792,43.637,158.174
C06176=1031.439,93.636,401.715,168.795,43.635,158.174
C06177=1031.445,93.885,401.696,168.796,43.633,158.174
C06178=1031.451,94.134,401.677,168.799,43.632,158.174
C06179=1031.457,94.383,401.658,168.802,43.630,158.174
C06180=1031.464,94.633,401.639,168.804,43.629,158.174
C06181=1031.469,94.882,401.620,168.806,43.627,158.174
C06182=1031.476,95.131,401.602,168.809,43.625,158.174
C06183=1031.482,95.380,401.582,168.811,43.624,158.174
C06184=1031.488,95.629,401.563,168.813,43.622,158.173
C06185=1031.494,95.878,401.544,168.816,43.620,158.173
C06186=1031.500,96.128,401.525,168.818,43.619,158.173
C06187=1031.507,96.377,401.506,168.820,43.618,158.173
C06188=1031.512,96.626,401.487,168.823,43.616,158.173
C06189=1031.519,96.875,401.468,168.825,43.615,158.173
C06190=1031.525,97.124,401.449,168.827,43.613,158.173
C06191=1031.532,97.374,401.429,168.830,43.612,158.173
C06192=1031.537,97.623,401.410,168.832,43.610,158.173
C06193=1031.544,97.872,401.392,168.834,43.608,158.172
C06194=1031.550,98.122,401.372,168.837,43.607,158.172
C06195=1031.556,98.370,401.353,168.840,43.605,158.172
C06196=1031.562,98.620,401.334,168.841,43.603,158.172
C06197=1031.568,98.869,401.315,168.844,43.602,158.172
C06198=1031.574,99.118,401.296,168.847,43.600,158.172
C06199=1031.581,99.367,401.276,168.848,43.599,158.172
C06200=1031.587,99.616,401.258,168.851,43.597,158.172
C06201=1031.593,99.865,401.239,168.854,43.595,158.172
C06202=1031.599,100.116,401.219,168.856,43.594,158.171
C06203=1031.606,100.364,401.200,168.858,43.593,158.171
C06204=1031.612,100.613,401.180,168.861,43.591,158.171
C06205=1031.617,100.863,401.161,168.863,43.590,158.171
C06206=1031.623,101.112,401.141,168.865,43.588,158.171
C06207=1031.630,101.361,401.123,168.868,43.587,158.171
C06208=1031.635,101.610,401.103,168.870,43.585,158.171
C06209=1031.641,101.859,401.083,168.873,43.584,158.171
C06210=1031.647,102.109,401.064,168.875,43.582,158.171
C06211=1031.654,102.357,401.045,168.877,43.581,158.171
C06212=1031.660,102.607,401.025,168.880,43.579,158.171
C06213=1031.666,102.856,401.005,168.883,43.578,158.171
C06214=1031.673,103.105,400.987,168.884,43.576,158.170
C06215=1031.678,103.355,400.967,168.887,43.575,158.170
C06216=1031.684,103.603,400.947,168.890,43.573,158.170
C06217=1031.690,103.853,400.928,168.891,43.572,158.170
C06218=1031.697,104.101,400.909,168.894,43.570,158.170
C06219=1031.702,104.351,400.889,168.897,43.568,158.170
C06220=1031.709,104.600,400.869,168.899,43.567,158.170
C06221=1031.715,104.850,400.850,168.901,43.565,158.170
C06222=1031.721,105.098,400.831,168.904,43.564,158.170
C06223=1031.727,105.348,400.811,168.907,43.562,158.170
C06224=1031.733,105.596,400.791,168.908,43.561,158.169
C06225=1031.739,105.846,400.772,168.911,43.560,158.169
C06226=1031.746,106.095,400.752,168.914,43.558,158.169
C06227=1031.752,106.344,400.733,168.915,43.557,158.169
C06228=1031.758,106.593,400.713,168.918,43.555,158.169
C06229=1031.763,106.843,400.694,168.921,43.554,158.169
C06230=1031.770,107.091,400.675,168.923,43.552,158.169
C06231=1031.776,107.341,400.655,168.925,43.551,158.169
C06232=1031.782,107.590,400.635,168.928,43.549,158.169
C06233=1031.788,107.840,400.616,168.931,43.547,158.168
C06234=1031.795,108.124,400.593,168.933,43.546,158.168
C06235=1031.803,108.410,400.571,168.936,43.544,158.168
C06236=1031.810,108.695,400.548,168.939,43.542,158.168
C06237=1031.816,108.981,400.526,168.941,43.540,158.168
C06238=1031.823,109.229,400.506,168.944,43.539,158.168
C06239=1031.829,109.479,400.487,168.947,43.537,158.168
C06240=1031.835,109.728,400.467,168.948,43.535,158.168
C06241=1031.841,109.977,400.447,168.951,43.534,158.168
C06242=1031.847,110.226,400.428,168.954,43.532,158.168
C06243=1031.854,110.476,400.407,168.955,43.531,158.168
C06244=1031.860,110.724,400.388,168.958,43.530,158.167
C06245=1031.866,110.974,400.369,168.961,43.528,158.167
C06246=1031.872,111.223,400.349,168.964,43.527,158.167
C06247=1031.879,111.472,400.328,168.965,43.525,158.167
C06248=1031.884,111.722,400.309,168.968,43.524,158.167
C06249=1031.890,111.970,400.289,168.971,43.522,158.167
C06250=1031.896,112.219,400.269,168.972,43.521,158.167
C06251=1031.903,112.469,400.249,168.975,43.520,158.167
C06252=1031.909,112.718,400.230,168.978,43.518,158.167
C06253=1031.914,112.967,400.210,168.980,43.516,158.167
C06254=1031.921,113.216,400.189,168.982,43.515,158.166
C06255=1031.927,113.465,400.169,168.985,43.514,158.166
C06256=1031.933,113.714,400.149,168.988,43.512,158.166
C06257=1031.938,113.964,400.130,168.990,43.511,158.166
C06258=1031.945,114.213,400.109,168.992,43.510,158.166
C06259=1031.951,114.462,400.089,168.995,43.508,158.166
C06260=1031.957,114.711,400.069,168.997,43.507,158.166
C06261=1031.963,114.960,400.049,168.999,43.505,158.166
C06262=1031.968,115.210,400.029,169.002,43.504,158.166
C06263=1031.974,115.458,400.009,169.004,43.503,158.166
C06264=1031.980,115.707,399.989,169.007,43.501,158.166
C06265=1031.986,115.956,399.969,169.010,43.500,158.166
C06266=1031.992,116.206,399.948,169.011,43.498,158.166
C06267=1031.998,116.455,399.928,169.014,43.497,158.166
C06268=1032.004,116.704,399.908,169.017,43.496,158.166
C06269=1032.011,116.953,399.887,169.019,43.494,158.165
C06270=1032.017,117.202,399.868,169.021,43.493,158.165
C06271=1032.022,117.452,399.848,169.024,43.491,158.165
C06272=1032.028,117.700,399.828,169.027,43.490,158.165
C06273=1032.034,117.950,399.807,169.029,43.489,158.165
C06274=1032.040,118.199,399.787,169.031,43.487,158.165
C06275=1032.046,118.448,399.767,169.034,43.486,158.165
C06276=1032.052,118.697,399.747,169.037,43.484,158.165
C06277=1032.058,118.946,399.727,169.038,43.483,158.165
C06278=1032.065,119.194,399.706,169.041,43.481,158.165
C06279=1032.071,119.444,399.686,169.044,43.480,158.165
C06280=1032.076,119.693,399.665,169.046,43.479,158.165
C06281=1032.082,119.942,399.645,169.048,43.477,158.164
C06282=1032.089,120.191,399.625,169.051,43.476,158.164
C06283=1032.095,120.440,399.605,169.054,43.474,158.164
C06284=1032.101,120.690,399.584,169.056,43.473,158.164
C06285=1032.107,120.939,399.564,169.058,43.471,158.164
C06286=1032.113,121.188,399.544,169.061,43.470,158.164
C06287=1032.119,121.437,399.524,169.064,43.468,158.164
C06288=1032.125,121.686,399.503,169.065,43.467,158.164
C06289=1032.131,121.935,399.483,169.068,43.466,158.164
C06290=1032.137,122.185,399.463,169.071,43.464,158.164
C06291=1032.144,122.433,399.442,169.074,43.463,158.164
C06292=1032.149,122.683,399.421,169.075,43.461,158.164
C06293=1032.155,122.931,399.401,169.078,43.460,158.164
C06294=1032.162,123.181,399.381,169.081,43.459,158.164
C06295=1032.168,123.430,399.361,169.084,43.457,158.163
C06296=1032.173,123.679,399.340,169.085,43.456,158.163
C06297=1032.180,123.928,399.320,169.088,43.454,158.163
C06298=1032.187,124.214,399.296,169.091,43.452,158.163
C06299=1032.194,124.498,399.274,169.093,43.451,158.163
C06300=1032.201,124.784,399.250,169.097,43.449,158.163
C06301=1032.208,125.069,399.226,169.100,43.447,158.163
C06302=1032.214,125.318,399.206,169.103,43.446,158.163
C06303=1032.221,125.567,399.186,169.104,43.445,158.163
C06304=1032.226,125.816,399.165,169.107,43.443,158.163
C06305=1032.233,126.065,399.145,169.110,43.442,158.163
C06306=1032.239,126.314,399.125,169.112,43.440,158.162
C06307=1032.245,126.564,399.104,169.114,43.439,158.162
C06308=1032.251,126.812,399.083,169.117,43.437,158.162
C06309=1032.258,127.062,399.063,169.120,43.436,158.162
C06310=1032.264,127.310,399.043,169.122,43.434,158.162
C06311=1032.269,127.560,399.022,169.125,43.433,158.162
C06312=1032.276,127.808,399.001,169.127,43.431,158.162
C06313=1032.282,128.058,398.981,169.130,43.430,158.162
C06314=1032.288,128.307,398.961,169.132,43.428,158.162
C06315=1032.294,128.556,398.939,169.135,43.427,158.162
C06316=1032.300,128.805,398.919,169.138,43.425,158.162
C06317=1032.307,129.054,398.899,169.139,43.424,158.161
C06318=1032.313,129.303,398.878,169.142,43.422,158.161
C06319=1032.319,129.552,398.857,169.145,43.421,158.161
C06320=1032.326,129.802,398.837,169.148,43.419,158.161
C06321=1032.332,130.050,398.816,169.150,43.418,158.161
C06322=1032.338,130.300,398.795,169.153,43.417,158.161
C06323=1032.344,130.549,398.775,169.155,43.415,158.161
C06324=1032.351,130.798,398.754,169.158,43.414,158.161
C06325=1032.356,131.047,398.734,169.160,43.412,158.161
C06326=1032.362,131.296,398.712,169.163,43.411,158.161
C06327=1032.368,131.545,398.692,169.166,43.410,158.161
C06328=1032.374,131.794,398.671,169.168,43.408,158.161
C06329=1032.380,132.043,398.651,169.170,43.407,158.161
C06330=1032.387,132.292,398.629,169.173,43.406,158.161
C06331=1032.392,132.541,398.608,169.176,43.404,158.160
C06332=1032.399,132.790,398.587,169.178,43.403,158.160
C06333=1032.405,133.040,398.567,169.180,43.402,158.160
C06334=1032.411,133.288,398.546,169.183,43.400,158.160
C06335=1032.417,133.538,398.525,169.186,43.399,158.160
C06336=1032.422,133.786,398.504,169.189,43.397,158.160
C06337=1032.429,134.035,398.483,169.191,43.396,158.160
C06338=1032.434,134.284,398.462,169.193,43.395,158.160
C06339=1032.441,134.533,398.441,169.196,43.393,158.160
C06340=1032.447,134.783,398.420,169.199,43.392,158.160
C06341=1032.453,135.032,398.399,169.201,43.390,158.160
C06342=1032.460,135.280,398.378,169.203,43.389,158.160
C06343=1032.465,135.530,398.357,169.206,43.388,158.160
C06344=1032.471,135.779,398.336,169.209,43.386,158.160
C06345=1032.478,136.028,398.315,169.212,43.385,158.160
C06346=1032.483,136.277,398.294,169.214,43.384,158.160
C06347=1032.490,136.526,398.273,169.217,43.382,158.159
C06348=1032.495,136.775,398.252,169.219,43.381,158.159
C06349=1032.502,137.024,398.231,169.222,43.380,158.159
C06350=1032.508,137.273,398.210,169.224,43.378,158.159
C06351=1032.514,137.522,398.189,169.227,43.377,158.159
C06352=1032.520,137.771,398.168,169.230,43.376,158.159
C06353=1032.526,138.020,398.146,169.232,43.374,158.159
C06354=1032.532,138.269,398.125,169.234,43.373,158.159
C06355=1032.538,138.518,398.104,169.237,43.372,158.159
C06356=1032.544,138.768,398.083,169.240,43.370,158.159
C06357=1032.551,139.016,398.062,169.243,43.369,158.159
C06358=1032.557,139.265,398.040,169.245,43.367,158.159
C06359=1032.562,139.514,398.019,169.247,43.366,158.159
C06360=1032.568,139.763,397.998,169.250,43.365,158.159
C06361=1032.574,140.013,397.977,169.253,43.363,158.159
C06362=1032.582,140.297,397.952,169.256,43.362,158.159
C06363=1032.588,140.582,397.927,169.258,43.361,158.159
C06364=1032.595,140.868,397.904,169.262,43.359,158.159
C06365=1032.602,141.153,397.879,169.265,43.358,158.159
C06366=1032.608,141.401,397.858,169.268,43.357,158.159
C06367=1032.614,141.650,397.836,169.270,43.355,158.158
C06368=1032.621,141.900,397.815,169.272,43.354,158.158
C06369=1032.626,142.148,397.793,169.275,43.353,158.158
C06370=1032.632,142.398,397.772,169.278,43.351,158.158
C06371=1032.638,142.647,397.751,169.280,43.350,158.158
C06372=1032.644,142.896,397.730,169.283,43.348,158.158
C06373=1032.650,143.145,397.708,169.286,43.347,158.158
C06374=1032.657,143.394,397.687,169.289,43.346,158.158
C06375=1032.663,143.643,397.665,169.291,43.345,158.158
C06376=1032.668,143.891,397.644,169.293,43.343,158.158
C06377=1032.675,144.141,397.622,169.296,43.342,158.158
C06378=1032.681,144.390,397.601,169.299,43.341,158.158
C06379=1032.687,144.639,397.579,169.302,43.340,158.158
C06380=1032.692,144.887,397.558,169.304,43.338,158.158
C06381=1032.699,145.137,397.536,169.307,43.337,158.158
C06382=1032.705,145.386,397.515,169.309,43.336,158.158
C06383=1032.712,145.635,397.493,169.312,43.334,158.158
C06384=1032.717,145.883,397.472,169.315,43.333,158.158
C06385=1032.723,146.133,397.451,169.317,43.331,158.157
C06386=1032.730,146.382,397.429,169.320,43.330,158.157
C06387=1032.736,146.631,397.407,169.323,43.329,158.157
C06388=1032.741,146.879,397.386,169.326,43.328,158.157
C06389=1032.747,147.129,397.364,169.329,43.327,158.157
C06390=1032.754,147.378,397.343,169.330,43.325,158.157
C06391=1032.760,147.627,397.321,169.333,43.324,158.157
C06392=1032.766,147.876,397.299,169.336,43.323,158.157
C06393=1032.772,148.124,397.278,169.339,43.321,158.157
C06394=1032.778,148.373,397.256,169.342,43.320,158.157
C06395=1032.783,148.623,397.234,169.344,43.319,158.157
C06396=1032.790,148.872,397.212,169.347,43.318,158.157
C06397=1032.796,149.121,397.190,169.350,43.316,158.157
C06398=1032.802,149.369,397.168,169.353,43.315,158.157
C06399=1032.808,149.618,397.147,169.355,43.314,158.157
C06400=1032.814,149.868,397.125,169.357,43.313,158.157
C06401=1032.820,150.117,397.103,169.360,43.312,158.157
C06402=1032.827,150.365,397.081,169.363,43.310,158.157
C06403=1032.831,150.614,397.059,169.366,43.309,158.157
C06404=1032.838,150.863,397.038,169.369,43.308,158.157
C06405=1032.844,151.113,397.016,169.372,43.307,158.157
C06406=1032.850,151.361,396.994,169.374,43.306,158.157
C06407=1032.856,151.610,396.972,169.377,43.304,158.157
C06408=1032.863,151.860,396.950,169.379,43.303,158.157
C06409=1032.867,152.108,396.929,169.382,43.302,158.157
C06410=1032.874,152.357,396.906,169.385,43.300,158.157
C06411=1032.880,152.606,396.885,169.387,43.299,158.157
C06412=1032.886,152.855,396.863,169.390,43.298,158.157
C06413=1032.893,153.104,396.841,169.393,43.297,158.157
C06414=1032.899,153.353,396.819,169.396,43.296,158.157
C06415=1032.905,153.602,396.797,169.399,43.295,158.157
C06416=1032.911,153.851,396.774,169.401,43.293,158.156
C06417=1032.916,154.100,396.753,169.404,43.292,158.156
C06418=1032.923,154.348,396.731,169.407,43.290,158.156
C06419=1032.929,154.598,396.709,169.409,43.289,158.156
C06420=1032.934,154.847,396.687,169.412,43.288,158.156
C06421=1032.941,155.096,396.664,169.414,43.287,158.156
C06422=1032.947,155.345,396.643,169.417,43.286,158.156
C06423=1032.953,155.594,396.620,169.420,43.285,158.156
C06424=1032.959,155.843,396.598,169.423,43.284,158.156
C06425=1032.965,156.092,396.576,169.426,43.282,158.156
C06426=1032.972,156.377,396.551,169.429,43.281,158.156
C06427=1032.979,156.661,396.525,169.432,43.280,158.156
C06428=1032.985,156.946,396.500,169.435,43.279,158.156
C06429=1032.992,157.231,396.475,169.438,43.277,158.156
C06430=1032.999,157.479,396.452,169.441,43.276,158.156
C06431=1033.005,157.728,396.431,169.444,43.274,158.156
C06432=1033.011,157.977,396.408,169.446,43.273,158.156
C06433=1033.017,158.227,396.386,169.449,43.272,158.156
C06434=1033.023,158.475,396.364,169.452,43.271,158.156
C06435=1033.029,158.725,396.341,169.455,43.270,158.156
C06436=1033.035,158.973,396.319,169.458,43.269,158.156
C06437=1033.041,159.222,396.297,169.461,43.267,158.156
C06438=1033.047,159.471,396.275,169.463,43.266,158.156
C06439=1033.053,159.720,396.252,169.466,43.265,158.156
C06440=1033.059,159.969,396.230,169.469,43.264,158.156
C06441=1033.065,160.218,396.207,169.472,43.263,158.156
C06442=1033.071,160.467,396.185,169.475,43.262,158.156
C06443=1033.076,160.715,396.162,169.478,43.261,158.156
C06444=1033.082,160.965,396.140,169.481,43.260,158.156
C06445=1033.088,161.213,396.118,169.483,43.259,158.156
C06446=1033.094,161.462,396.095,169.485,43.258,158.156
C06447=1033.100,161.711,396.072,169.488,43.257,158.156
C06448=1033.105,161.960,396.049,169.491,43.256,158.156
C06449=1033.111,162.209,396.027,169.494,43.255,158.156
C06450=1033.117,162.458,396.004,169.497,43.254,158.156
C06451=1033.123,162.707,395.981,169.500,43.253,158.156
C06452=1033.129,162.956,395.958,169.503,43.252,158.156
C06453=1033.135,163.204,395.936,169.505,43.251,158.156
C06454=1033.141,163.453,395.913,169.508,43.250,158.156
C06455=1033.146,163.703,395.891,169.511,43.248,158.156
C06456=1033.152,163.952,395.868,169.514,43.248,158.156
C06457=1033.158,164.200,395.845,169.517,43.247,158.156
C06458=1033.164,164.449,395.822,169.520,43.245,158.156
C06459=1033.170,164.698,395.799,169.523,43.244,158.156
C06460=1033.176,164.947,395.777,169.526,43.244,158.156
C06461=1033.181,165.196,395.754,169.529,43.243,158.156
C06462=1033.188,165.444,395.731,169.531,43.241,158.156
C06463=1033.194,165.693,395.708,169.534,43.240,158.156
C06464=1033.199,165.942,395.685,169.536,43.239,158.156
C06465=1033.205,166.191,395.662,169.539,43.239,158.157
C06466=1033.212,166.440,395.640,169.542,43.238,158.156
C06467=1033.217,166.689,395.617,169.545,43.236,158.156
C06468=1033.223,166.937,395.594,169.548,43.235,158.156
C06469=1033.229,167.187,395.571,169.550,43.234,158.156
C06470=1033.236,167.436,395.548,169.553,43.233,158.157
C06471=1033.242,167.685,395.526,169.556,43.232,158.157
C06472=1033.247,167.933,395.503,169.559,43.231,158.157
C06473=1033.253,168.182,395.480,169.562,43.230,158.157
C06474=1033.259,168.431,395.457,169.565,43.229,158.157
C06475=1033.265,168.680,395.434,169.568,43.228,158.157
C06476=1033.271,168.929,395.411,169.571,43.227,158.157
C06477=1033.277,169.178,395.388,169.573,43.226,158.157
C06478=1033.283,169.427,395.365,169.578,43.225,158.157
C06479=1033.289,169.676,395.342,169.580,43.224,158.157
C06480=1033.295,169.925,395.320,169.583,43.223,158.157
C06481=1033.301,170.174,395.297,169.586,43.222,158.157
C06482=1033.307,170.423,395.274,169.589,43.221,158.157
C06483=1033.312,170.671,395.251,169.592,43.220,158.157
C06484=1033.318,170.920,395.227,169.595,43.219,158.157
C06485=1033.325,171.169,395.205,169.598,43.218,158.157
C06486=1033.331,171.418,395.182,169.600,43.217,158.157
C06487=1033.337,171.667,395.159,169.603,43.216,158.157
C06488=1033.343,171.916,395.136,169.606,43.215,158.157
C06489=1033.348,172.165,395.113,169.609,43.214,158.157
C06490=1033.356,172.448,395.086,169.612,43.212,158.157
C06491=1033.363,172.733,395.060,169.616,43.211,158.157
C06492=1033.370,173.017,395.034,169.620,43.210,158.157
C06493=1033.377,173.302,395.007,169.623,43.209,158.157
C06494=1033.382,173.550,394.984,169.625,43.208,158.157
C06495=1033.389,173.799,394.962,169.628,43.207,158.157
C06496=1033.395,174.049,394.938,169.631,43.206,158.157
C06497=1033.401,174.297,394.915,169.634,43.205,158.157
C06498=1033.407,174.546,394.892,169.637,43.204,158.157
C06499=1033.413,174.795,394.869,169.641,43.203,158.157
C06500=1033.420,175.044,394.846,169.644,43.202,158.157
C06501=1033.426,175.292,394.822,169.647,43.201,158.157
C06502=1033.432,175.541,394.800,169.650,43.200,158.157
C06503=1033.438,175.791,394.776,169.652,43.199,158.157
C06504=1033.444,176.039,394.753,169.655,43.198,158.157
C06505=1033.450,176.288,394.730,169.658,43.197,158.157
C06506=1033.456,176.536,394.707,169.661,43.196,158.157
C06507=1033.463,176.785,394.683,169.664,43.195,158.157
C06508=1033.469,177.034,394.660,169.668,43.194,158.158
C06509=1033.474,177.283,394.637,169.671,43.193,158.158
C06510=1033.481,177.532,394.613,169.674,43.192,158.158
C06511=1033.487,177.781,394.590,169.676,43.190,158.158
C06512=1033.493,178.029,394.567,169.679,43.190,158.158
C06513=1033.500,178.279,394.544,169.682,43.189,158.158
C06514=1033.505,178.528,394.521,169.685,43.188,158.158
C06515=1033.512,178.776,394.497,169.689,43.187,158.158
C06516=1033.518,179.025,394.474,169.692,43.186,158.158
C06517=1033.524,179.274,394.450,169.695,43.185,158.158
C06518=1033.530,179.523,394.427,169.698,43.183,158.158
C06519=1033.537,179.771,394.404,169.701,43.183,158.158
C06520=1033.543,180.020,394.381,169.704,43.182,158.158
C06521=1033.549,180.269,394.357,169.707,43.180,158.158
C06522=1033.555,180.518,394.334,169.710,43.180,158.158
C06523=1033.561,180.766,394.310,169.713,43.179,158.158
C06524=1033.567,181.016,394.287,169.716,43.177,158.158
C06525=1033.573,181.264,394.263,169.719,43.177,158.158
C06526=1033.581,181.514,394.241,169.722,43.176,158.158
C06527=1033.587,181.762,394.217,169.726,43.174,158.158
C06528=1033.593,182.011,394.194,169.729,43.173,158.158
C06529=1033.599,182.260,394.170,169.732,43.173,158.158
C06530=1033.608,182.616,394.137,169.737,43.171,158.158
C06531=1033.617,182.971,394.103,169.740,43.170,158.158
C06532=1033.626,183.328,394.070,169.745,43.168,158.158
C06533=1033.634,183.684,394.035,169.749,43.168,158.159
C06534=1033.640,183.932,394.011,169.752,43.166,158.159
C06535=1033.645,184.180,393.987,169.756,43.166,158.159
C06536=1033.652,184.429,393.963,169.759,43.165,158.159
C06537=1033.657,184.679,393.940,169.762,43.164,158.159
C06538=1033.664,184.928,393.916,169.765,43.164,158.159
C06539=1033.669,185.176,393.891,169.768,43.162,158.159
C06540=1033.675,185.424,393.868,169.771,43.162,158.159
C06541=1033.682,185.673,393.844,169.774,43.161,158.159
C06542=1033.687,185.922,393.819,169.777,43.160,158.159
C06543=1033.694,186.171,393.795,169.781,43.159,158.159
C06544=1033.699,186.420,393.771,169.784,43.159,158.159
C06545=1033.705,186.668,393.748,169.787,43.158,158.159
C06546=1033.711,186.918,393.723,169.790,43.157,158.160
C06547=1033.717,187.166,393.700,169.793,43.157,158.160
C06548=1033.722,187.415,393.675,169.796,43.156,158.160
C06549=1033.728,187.664,393.652,169.800,43.155,158.160
C06550=1033.733,187.876,393.631,169.802,43.155,158.160
C06551=1033.739,188.089,393.610,169.805,43.153,158.160
C06552=1033.744,188.302,393.589,169.808,43.153,158.160
C06553=1033.749,188.515,393.569,169.811,43.152,158.160
C06554=1033.755,188.728,393.548,169.813,43.152,158.160
C06555=1033.760,188.941,393.527,169.816,43.151,158.160
C06556=1033.764,189.153,393.507,169.819,43.150,158.160
C06557=1033.770,189.366,393.486,169.821,43.150,158.160
C06558=1033.776,189.615,393.462,169.824,43.149,158.160
C06559=1033.782,189.863,393.438,169.827,43.148,158.161
C06560=1033.788,190.113,393.413,169.831,43.148,158.161
C06561=1033.794,190.361,393.390,169.833,43.146,158.161
C06562=1033.800,190.610,393.365,169.837,43.146,158.161
C06563=1033.806,190.858,393.341,169.840,43.145,158.161
C06564=1033.812,191.108,393.317,169.844,43.145,158.161
C06565=1033.818,191.356,393.293,169.846,43.144,158.161
C06566=1033.824,191.605,393.268,169.849,43.143,158.161
C06567=1033.830,191.854,393.244,169.853,43.142,158.161
C06568=1033.836,192.102,393.219,169.856,43.141,158.161
C06569=1033.843,192.351,393.195,169.859,43.141,158.162
C06570=1033.848,192.600,393.171,169.862,43.140,158.162
C06571=1033.855,192.849,393.147,169.866,43.139,158.162
C06572=1033.860,193.097,393.123,169.869,43.138,158.162
C06573=1033.866,193.346,393.099,169.872,43.138,158.162
C06574=1033.873,193.595,393.074,169.876,43.137,158.162
C06575=1033.879,193.843,393.050,169.879,43.136,158.162
C06576=1033.885,194.093,393.025,169.882,43.135,158.162
C06577=1033.891,194.342,393.001,169.885,43.135,158.162
C06578=1033.897,194.590,392.977,169.889,43.134,158.163
C06579=1033.903,194.838,392.952,169.892,43.134,158.163
C06580=1033.909,195.088,392.928,169.895,43.132,158.163
C06581=1033.915,195.336,392.904,169.899,43.132,158.163
C06582=1033.922,195.585,392.879,169.902,43.131,158.163
C06583=1033.928,195.834,392.855,169.905,43.131,158.163
C06584=1033.934,196.082,392.830,169.908,43.129,158.163
C06585=1033.940,196.331,392.806,169.912,43.129,158.163
C06586=1033.946,196.580,392.781,169.915,43.128,158.163
C06587=1033.952,196.828,392.757,169.918,43.128,158.163
C06588=1033.958,197.077,392.733,169.922,43.126,158.163
C06589=1033.965,197.326,392.708,169.925,43.126,158.164
C06590=1033.971,197.574,392.684,169.928,43.125,158.164
C06591=1033.978,197.823,392.659,169.932,43.125,158.164
C06592=1033.983,198.072,392.634,169.935,43.124,158.164
C06593=1033.990,198.321,392.610,169.938,43.123,158.164
C06594=1033.996,198.569,392.585,169.942,43.122,158.164
C06595=1034.002,198.818,392.561,169.945,43.122,158.164
C06596=1034.009,199.067,392.536,169.948,43.121,158.164
C06597=1034.014,199.316,392.511,169.952,43.121,158.165
C06598=1034.021,199.564,392.487,169.955,43.120,158.165
C06599=1034.027,199.813,392.462,169.958,43.119,158.165
C06600=1034.034,200.061,392.438,169.962,43.118,158.165
C06601=1034.040,200.311,392.413,169.965,43.118,158.165
C06602=1034.046,200.560,392.389,169.969,43.117,158.165
C06603=1034.052,200.808,392.364,169.972,43.116,158.165
C06604=1034.058,201.056,392.339,169.975,43.116,158.165
C06605=1034.064,201.305,392.314,169.979,43.115,158.166
C06606=1034.070,201.554,392.289,169.982,43.115,158.166
C06607=1034.077,201.802,392.264,169.985,43.114,158.166
C06608=1034.082,202.051,392.240,169.990,43.113,158.166
C06609=1034.089,202.300,392.214,169.993,43.113,158.166
C06610=1034.095,202.548,392.189,169.996,43.112,158.166
C06611=1034.101,202.798,392.164,170.000,43.112,158.166
C06612=1034.107,203.046,392.139,170.003,43.111,158.167
C06613=1034.112,203.294,392.114,170.006,43.111,158.167
C06614=1034.118,203.544,392.089,170.010,43.110,158.167
C06615=1034.125,203.792,392.064,170.013,43.109,158.167
C06616=1034.131,204.041,392.039,170.017,43.109,158.167
C06617=1034.138,204.289,392.014,170.020,43.108,158.167
C06618=1034.163,205.339,391.908,170.348,43.213,158.214
C06619=1034.172,205.681,391.872,170.352,43.213,158.215
C06620=1034.182,206.022,391.836,170.355,43.214,158.215
C06621=1034.191,206.362,391.800,170.358,43.214,158.215
C06622=1034.200,206.704,391.764,170.361,43.214,158.216
C06623=1034.207,206.952,391.738,170.365,43.214,158.216
C06624=1034.214,207.200,391.711,170.367,43.214,158.216
C06625=1034.221,207.449,391.684,170.369,43.214,158.216
C06626=1034.227,207.697,391.658,170.371,43.215,158.217
C06627=1034.234,207.946,391.631,170.375,43.215,158.217
C06628=1034.241,208.195,391.605,170.377,43.215,158.217
C06629=1034.247,208.443,391.578,170.379,43.215,158.217
C06630=1034.254,208.692,391.552,170.381,43.216,158.218
C06631=1034.261,208.940,391.526,170.385,43.216,158.218
C06632=1034.268,209.189,391.499,170.387,43.216,158.218
C06633=1034.274,209.438,391.472,170.389,43.216,158.218
C06634=1034.281,209.685,391.445,170.391,43.217,158.219
C06635=1034.288,209.934,391.419,170.395,43.217,158.219
C06636=1034.295,210.183,391.392,170.397,43.217,158.219
C06637=1034.301,210.431,391.366,170.399,43.217,158.219
C06638=1034.308,210.680,391.339,170.402,43.217,158.220
C06639=1034.315,210.928,391.312,170.405,43.218,158.220
C06640=1034.321,211.176,391.286,170.407,43.218,158.220
C06641=1034.328,211.425,391.259,170.409,43.218,158.220
C06642=1034.335,211.674,391.232,170.412,43.218,158.221
C06643=1034.341,211.922,391.205,170.415,43.219,158.221
C06644=1034.348,212.171,391.178,170.417,43.219,158.221
C06645=1034.354,212.420,391.151,170.419,43.220,158.221
C06646=1034.361,212.667,391.125,170.422,43.220,158.222
C06647=1034.368,212.916,391.098,170.425,43.220,158.222
C06648=1034.375,213.165,391.071,170.427,43.220,158.222
C06649=1034.381,213.413,391.044,170.430,43.220,158.222
C06650=1034.388,213.661,391.017,170.432,43.221,158.223
C06651=1034.394,213.911,390.990,170.435,43.221,158.223
C06652=1034.401,214.158,390.964,170.438,43.221,158.223
C06653=1034.407,214.407,390.937,170.440,43.221,158.223
C06654=1034.415,214.656,390.910,170.442,43.222,158.224
C06655=1034.421,214.904,390.883,170.445,43.222,158.224
C06656=1034.428,215.152,390.856,170.448,43.222,158.224
C06657=1034.434,215.401,390.829,170.450,43.222,158.224
C06658=1034.442,215.649,390.802,170.453,43.223,158.225
C06659=1034.448,215.898,390.775,170.456,43.223,158.225
C06660=1034.455,216.146,390.749,170.458,43.224,158.225
C06661=1034.461,216.395,390.722,170.460,43.224,158.225
C06662=1034.469,216.643,390.694,170.464,43.224,158.226
C06663=1034.475,216.892,390.667,170.466,43.224,158.226
C06664=1034.482,217.140,390.641,170.468,43.225,158.226
C06665=1034.488,217.389,390.614,170.471,43.225,158.226
C06666=1034.496,217.637,390.586,170.474,43.225,158.227
C06667=1034.502,217.886,390.559,170.477,43.225,158.227
C06668=1034.509,218.134,390.532,170.479,43.225,158.227
C06669=1034.515,218.382,390.506,170.481,43.226,158.227
C06670=1034.523,218.631,390.479,170.485,43.226,158.228
C06671=1034.529,218.880,390.452,170.487,43.226,158.228
C06672=1034.536,219.128,390.424,170.489,43.227,158.228
C06673=1034.543,219.376,390.397,170.492,43.227,158.229
C06674=1034.549,219.625,390.370,170.495,43.227,158.229
C06675=1034.559,219.971,390.331,170.498,43.227,158.229
C06676=1034.568,220.318,390.294,170.502,43.228,158.230
C06677=1034.577,220.666,390.256,170.506,43.229,158.230
C06678=1034.586,221.012,390.218,170.509,43.229,158.230
C06679=1034.593,221.260,390.190,170.513,43.229,158.231
C06680=1034.599,221.510,390.163,170.515,43.230,158.231
C06681=1034.606,221.757,390.136,170.517,43.230,158.231
C06682=1034.613,222.005,390.108,170.520,43.230,158.231
C06683=1034.620,222.254,390.081,170.523,43.230,158.232
C06684=1034.626,222.503,390.054,170.525,43.231,158.232
C06685=1034.633,222.751,390.026,170.528,43.231,158.232
C06686=1034.640,222.999,389.999,170.531,43.232,158.233
C06687=1034.646,223.247,389.971,170.534,43.232,158.233
C06688=1034.653,223.496,389.944,170.536,43.232,158.233
C06689=1034.659,223.745,389.917,170.538,43.232,158.233
C06690=1034.666,223.993,389.889,170.542,43.233,158.234
C06691=1034.673,224.242,389.861,170.544,43.233,158.234
C06692=1034.680,224.490,389.834,170.547,43.233,158.234
C06693=1034.687,224.738,389.806,170.549,43.234,158.234
C06694=1034.693,224.987,389.779,170.553,43.234,158.235
C06695=1034.700,225.236,389.752,170.555,43.235,158.235
C06696=1034.706,225.484,389.724,170.557,43.235,158.235
C06697=1034.713,225.732,389.697,170.561,43.235,158.236
C06698=1034.720,225.980,389.669,170.563,43.235,158.236
C06699=1034.727,226.228,389.642,170.566,43.235,158.236
C06700=1034.733,226.477,389.614,170.569,43.236,158.237
C06701=1034.740,226.725,389.586,170.572,43.236,158.237
C06702=1034.746,226.974,389.559,170.574,43.237,158.237
C06703=1034.754,227.223,389.532,170.576,43.237,158.237
C06704=1034.760,227.471,389.504,170.580,43.237,158.238
C06705=1034.767,227.719,389.476,170.582,43.238,158.238
C06706=1034.774,227.968,389.449,170.585,43.238,158.238
C06707=1034.781,228.216,389.421,170.587,43.238,158.238
C06708=1034.787,228.465,389.393,170.591,43.238,158.239
C06709=1034.794,228.713,389.366,170.593,43.239,158.239
C06710=1034.801,228.962,389.338,170.596,43.239,158.239
C06711=1034.807,229.210,389.310,170.599,43.240,158.240
C06712=1034.814,229.458,389.282,170.601,43.241,158.240
C06713=1034.821,229.706,389.254,170.604,43.241,158.240
C06714=1034.828,229.955,389.226,170.607,43.241,158.241
C06715=1034.834,230.203,389.198,170.610,43.242,158.241
C06716=1034.841,230.452,389.171,170.612,43.242,158.241
C06717=1034.847,230.700,389.142,170.616,43.242,158.241
C06718=1034.854,230.949,389.115,170.618,43.243,158.242
C06719=1034.860,231.197,389.087,170.621,43.243,158.242
C06720=1034.867,231.445,389.058,170.624,43.243,158.242
C06721=1034.874,231.694,389.031,170.627,43.243,158.243
C06722=1034.881,231.942,389.003,170.629,43.244,158.243
C06723=1034.887,232.190,388.975,170.632,43.244,158.243
C06724=1034.894,232.439,388.948,170.635,43.245,158.244
C06725=1034.900,232.687,388.919,170.637,43.245,158.244
C06726=1034.907,232.935,388.891,170.640,43.246,158.244
C06727=1034.914,233.184,388.863,170.643,43.246,158.245
C06728=1034.921,233.432,388.835,170.646,43.247,158.245
C06729=1034.927,233.680,388.806,170.649,43.247,158.245
C06730=1034.933,233.929,388.779,170.652,43.248,158.245
C06731=1034.942,234.268,388.741,170.655,43.248,158.246
C06732=1034.952,234.607,388.702,170.660,43.249,158.246
C06733=1034.960,234.947,388.663,170.663,43.250,158.247
C06734=1034.970,235.286,388.625,170.668,43.249,158.247
C06735=1034.976,235.534,388.597,170.670,43.250,158.248
C06736=1034.983,235.783,388.569,170.673,43.250,158.248
C06737=1034.990,236.030,388.541,170.676,43.251,158.248
C06738=1034.996,236.279,388.512,170.679,43.251,158.248
C06739=1035.003,236.528,388.485,170.681,43.252,158.249
C06740=1035.010,236.775,388.456,170.685,43.252,158.249
C06741=1035.017,237.025,388.428,170.687,43.253,158.249
C06742=1035.023,237.273,388.399,170.690,43.253,158.250
C06743=1035.030,237.521,388.371,170.693,43.254,158.250
C06744=1035.037,237.769,388.343,170.696,43.254,158.250
C06745=1035.044,238.017,388.315,170.698,43.255,158.251
C06746=1035.050,238.265,388.286,170.702,43.255,158.251
C06747=1035.056,238.514,388.258,170.705,43.255,158.251
C06748=1035.064,238.762,388.230,170.707,43.256,158.252
C06749=1035.070,239.011,388.201,170.711,43.256,158.252
C06750=1035.077,239.259,388.173,170.713,43.257,158.252
C06751=1035.084,239.507,388.145,170.716,43.257,158.253
C06752=1035.090,239.756,388.116,170.719,43.258,158.253
C06753=1035.097,240.004,388.088,170.722,43.258,158.253
C06754=1035.104,240.252,388.060,170.724,43.259,158.254
C06755=1035.111,240.500,388.031,170.728,43.259,158.254
C06756=1035.117,240.749,388.003,170.731,43.259,158.254
C06757=1035.124,240.997,387.974,170.733,43.260,158.255
C06758=1035.130,241.245,387.945,170.737,43.260,158.255
C06759=1035.136,241.494,387.917,170.739,43.261,158.255
C06760=1035.143,241.742,387.888,170.742,43.261,158.256
C06761=1035.150,241.990,387.859,170.745,43.262,158.256
C06762=1035.157,242.239,387.831,170.748,43.262,158.256
C06763=1035.163,242.487,387.802,170.751,43.263,158.257
C06764=1035.170,242.735,387.774,170.754,43.263,158.257
C06765=1035.176,242.983,387.745,170.757,43.264,158.257
C06766=1035.184,243.232,387.717,170.760,43.264,158.258
C06767=1035.190,243.480,387.688,170.763,43.265,158.258
C06768=1035.197,243.728,387.659,170.765,43.265,158.258
C06769=1035.203,243.976,387.630,170.769,43.266,158.259
C06770=1035.209,244.224,387.601,170.772,43.266,158.259
C06771=1035.217,244.474,387.573,170.774,43.267,158.259
C06772=1035.223,244.722,387.544,170.778,43.268,158.260
C06773=1035.230,244.969,387.516,170.780,43.268,158.260
C06774=1035.236,245.218,387.487,170.784,43.269,158.260
C06775=1035.243,245.466,387.457,170.787,43.269,158.261
C06776=1035.249,245.715,387.428,170.789,43.270,158.261
C06777=1035.255,245.963,387.399,170.793,43.270,158.261
C06778=1035.262,246.211,387.370,170.795,43.271,158.262
C06779=1035.269,246.459,387.342,170.799,43.271,158.262
C06780=1035.276,246.707,387.312,170.802,43.272,158.263
C06781=1035.282,246.956,387.283,170.804,43.273,158.263
C06782=1035.288,247.204,387.254,170.808,43.273,158.263
C06783=1035.294,247.452,387.225,170.810,43.274,158.264
C06784=1035.302,247.700,387.196,170.814,43.275,158.264
C06785=1035.308,247.949,387.167,170.817,43.275,158.264
C06786=1035.314,248.197,387.138,170.819,43.276,158.265
C06787=1035.323,248.530,387.099,170.824,43.277,158.265
C06788=1035.332,248.864,387.060,170.827,43.278,158.266
C06789=1035.341,249.197,387.020,170.832,43.278,158.266
C06790=1035.350,249.530,386.982,170.835,43.279,158.267
C06791=1035.356,249.779,386.953,170.839,43.280,158.267
C06792=1035.363,250.027,386.923,170.842,43.280,158.268
C06793=1035.369,250.276,386.894,170.845,43.281,158.268
C06794=1035.376,250.523,386.864,170.848,43.281,158.268
C06795=1035.383,250.772,386.836,170.852,43.282,158.269
C06796=1035.390,251.020,386.806,170.854,43.283,158.269
C06797=1035.396,251.268,386.777,170.857,43.283,158.269
C06798=1035.403,251.517,386.748,170.861,43.284,158.270
C06799=1035.409,251.764,386.718,170.863,43.284,158.270
C06800=1035.416,252.013,386.689,170.867,43.285,158.270
C06801=1035.423,252.261,386.660,170.870,43.285,158.271
C06802=1035.429,252.509,386.631,170.872,43.286,158.271
C06803=1035.437,252.757,386.601,170.876,43.287,158.272
C06804=1035.443,253.005,386.572,170.879,43.288,158.272
C06805=1035.450,253.254,386.543,170.882,43.288,158.272
C06806=1035.456,253.502,386.514,170.885,43.289,158.273
C06807=1035.462,253.750,386.484,170.888,43.289,158.273
C06808=1035.470,253.998,386.455,170.892,43.290,158.274
C06809=1035.476,254.246,386.426,170.894,43.290,158.274
C06810=1035.483,254.495,386.396,170.898,43.291,158.274
C06811=1035.490,254.743,386.367,170.901,43.292,158.275
C06812=1035.497,254.992,386.338,170.904,43.293,158.275
C06813=1035.503,255.239,386.308,170.907,43.293,158.275
C06814=1035.510,255.488,386.278,170.910,43.293,158.276
C06815=1035.517,255.735,386.249,170.914,43.294,158.276
C06816=1035.523,255.983,386.220,170.916,43.295,158.277
C06817=1035.530,256.232,386.191,170.919,43.295,158.277
C06818=1035.537,256.480,386.161,170.923,43.296,158.277
C06819=1035.544,256.728,386.132,170.926,43.296,158.278
C06820=1035.550,256.976,386.102,170.929,43.297,158.278
C06821=1035.557,257.225,386.073,170.932,43.298,158.278
C06822=1035.564,257.473,386.042,170.936,43.298,158.279
C06823=1035.571,257.721,386.014,170.939,43.299,158.279
C06824=1035.578,257.969,385.984,170.942,43.299,158.280
C06825=1035.585,258.217,385.955,170.945,43.300,158.280
C06826=1035.592,258.465,385.925,170.948,43.300,158.280
C06827=1035.598,258.714,385.896,170.952,43.301,158.281
C06828=1035.605,258.962,385.865,170.955,43.302,158.281
C06829=1035.611,259.210,385.836,170.958,43.303,158.281
C06830=1035.619,259.458,385.806,170.961,43.303,158.282
C06831=1035.625,259.707,385.777,170.964,43.303,158.282
C06832=1035.633,259.954,385.748,170.968,43.304,158.283
C06833=1035.640,260.203,385.718,170.971,43.305,158.283
C06834=1035.646,260.450,385.689,170.974,43.306,158.283
C06835=1035.653,260.699,385.658,170.977,43.306,158.284
C06836=1035.660,260.948,385.629,170.981,43.307,158.284
C06837=1035.667,261.195,385.599,170.984,43.307,158.285
C06838=1035.674,261.443,385.569,170.987,43.308,158.285
C06839=1035.680,261.691,385.540,170.991,43.309,158.285
C06840=1035.687,261.940,385.510,170.993,43.310,158.286
C06841=1035.694,262.188,385.480,170.997,43.310,158.286
C06842=1035.700,262.436,385.450,171.000,43.311,158.287
C06843=1035.710,262.768,385.409,171.005,43.312,158.287
C06844=1035.718,263.100,385.370,171.008,43.313,158.288
C06845=1035.727,263.432,385.330,171.013,43.314,158.288
C06846=1035.736,263.764,385.289,171.018,43.315,158.289
C06847=1035.742,264.012,385.259,171.021,43.316,158.289
C06848=1035.749,264.260,385.229,171.025,43.316,158.290
C06849=1035.757,264.508,385.199,171.027,43.317,158.290
C06850=1035.763,264.756,385.169,171.031,43.318,158.291
C06851=1035.770,265.004,385.138,171.034,43.319,158.291
C06852=1035.777,265.253,385.108,171.038,43.319,158.291
C06853=1035.783,265.500,385.078,171.041,43.320,158.292
C06854=1035.790,265.749,385.048,171.045,43.321,158.292
C06855=1035.797,265.997,385.018,171.047,43.322,158.293
C06856=1035.803,266.244,384.988,171.050,43.322,158.293
C06857=1035.811,266.493,384.958,171.054,43.323,158.294
C06858=1035.817,266.741,384.927,171.057,43.324,158.294
C06859=1035.824,266.989,384.897,171.061,43.324,158.294
C06860=1035.831,267.237,384.867,171.064,43.325,158.295
C06861=1035.837,267.485,384.836,171.068,43.327,158.295
C06862=1035.844,267.733,384.807,171.070,43.327,158.296
C06863=1035.850,267.981,384.776,171.074,43.328,158.296
C06864=1035.857,268.230,384.746,171.077,43.329,158.297
C06865=1035.864,268.478,384.714,171.081,43.329,158.297
C06866=1035.871,268.725,384.685,171.084,43.330,158.298
C06867=1035.878,268.973,384.655,171.088,43.331,158.298
C06868=1035.884,269.222,384.624,171.092,43.332,158.299
C06869=1035.891,269.470,384.594,171.095,43.333,158.299
C06870=1035.897,269.718,384.563,171.097,43.334,158.299
C06871=1035.905,269.965,384.533,171.101,43.334,158.300
C06872=1035.911,270.214,384.502,171.104,43.335,158.300
C06873=1035.918,270.462,384.472,171.108,43.336,158.301
C06874=1035.924,270.710,384.441,171.112,43.337,158.301
C06875=1035.931,270.958,384.411,171.115,43.338,158.302
C06876=1035.938,271.206,384.380,171.118,43.339,158.302
C06877=1035.945,271.454,384.350,171.122,43.339,158.303
C06878=1035.951,271.702,384.319,171.125,43.340,158.303
C06879=1035.958,271.950,384.288,171.128,43.341,158.304
C06880=1035.965,272.198,384.258,171.132,43.342,158.304
C06881=1035.971,272.446,384.226,171.135,43.343,158.304
C06882=1035.979,272.694,384.196,171.139,43.343,158.305
C06883=1035.985,272.942,384.165,171.142,43.345,158.305
C06884=1035.991,273.190,384.134,171.146,43.345,158.306
C06885=1035.999,273.438,384.104,171.149,43.346,158.306
C06886=1036.005,273.686,384.073,171.153,43.347,158.307
C06887=1036.012,273.934,384.042,171.156,43.348,158.307
C06888=1036.019,274.182,384.011,171.160,43.349,158.308
C06889=1036.025,274.430,383.980,171.163,43.350,158.308
C06890=1036.032,274.678,383.950,171.167,43.351,158.309
C06891=1036.039,274.926,383.919,171.170,43.352,158.309
C06892=1036.045,275.174,383.888,171.174,43.352,158.310
C06893=1036.052,275.422,383.857,171.177,43.354,158.310
C06894=1036.059,275.670,383.826,171.180,43.354,158.311
C06895=1036.066,275.918,383.795,171.184,43.356,158.311
C06896=1036.072,276.166,383.765,171.187,43.356,158.312
C06897=1036.079,276.414,383.734,171.191,43.357,158.312
C06898=1036.086,276.662,383.702,171.194,43.358,158.313
C06899=1036.095,276.999,383.660,171.199,43.360,158.313
C06900=1036.104,277.335,383.619,171.204,43.361,158.314
C06901=1036.113,277.672,383.576,171.208,43.362,158.314
C06902=1036.123,278.009,383.534,171.214,43.363,158.315
C06903=1036.130,278.257,383.503,171.218,43.364,158.316
C06904=1036.136,278.504,383.472,171.220,43.365,158.316
C06905=1036.143,278.752,383.440,171.224,43.366,158.317
C06906=1036.149,279.000,383.409,171.227,43.367,158.317
C06907=1036.156,279.249,383.378,171.231,43.368,158.318
C06908=1036.162,279.496,383.347,171.235,43.369,158.318
C06909=1036.169,279.744,383.315,171.238,43.370,158.319
C06910=1036.176,279.992,383.284,171.242,43.371,158.319
C06911=1036.183,280.240,383.253,171.245,43.372,158.320
C06912=1036.190,280.488,383.222,171.249,43.373,158.320
C06913=1036.197,280.736,383.190,171.253,43.374,158.321
C06914=1036.204,280.984,383.159,171.256,43.375,158.321
C06915=1036.210,281.231,383.127,171.260,43.376,158.322
C06916=1036.217,281.479,383.096,171.263,43.377,158.322
C06917=1036.223,281.728,383.065,171.267,43.378,158.323
C06918=1036.230,281.976,383.034,171.272,43.379,158.323
C06919=1036.237,282.224,383.002,171.275,43.380,158.324
C06920=1036.244,282.472,382.971,171.279,43.381,158.324
C06921=1036.250,282.720,382.940,171.282,43.382,158.325
C06922=1036.257,282.967,382.908,171.286,43.383,158.325
C06923=1036.264,283.215,382.876,171.290,43.385,158.326
C06924=1036.271,283.463,382.845,171.293,43.385,158.326
C06925=1036.278,283.710,382.813,171.297,43.386,158.327
C06926=1036.284,283.958,382.782,171.300,43.387,158.327
C06927=1036.291,284.206,382.750,171.304,43.388,158.328
C06928=1036.298,284.454,382.719,171.308,43.390,158.329
C06929=1036.305,284.703,382.687,171.311,43.390,158.329
C06930=1036.312,284.951,382.656,171.315,43.392,158.330
C06931=1036.318,285.199,382.624,171.318,43.392,158.330
C06932=1036.325,285.446,382.592,171.322,43.394,158.331
C06933=1036.332,285.694,382.561,171.326,43.395,158.331
C06934=1036.339,285.942,382.529,171.330,43.396,158.332
C06935=1036.346,286.190,382.498,171.334,43.397,158.332
C06936=1036.352,286.438,382.466,171.338,43.398,158.333
C06937=1036.360,286.686,382.434,171.341,43.399,158.333
C06938=1036.367,286.933,382.402,171.345,43.400,158.334
C06939=1036.373,287.181,382.371,171.348,43.401,158.334
C06940=1036.381,287.429,382.339,171.352,43.402,158.335
C06941=1036.386,287.677,382.307,171.356,43.403,158.335
C06942=1036.393,287.925,382.275,171.359,43.405,158.336
C06943=1036.400,288.172,382.243,171.364,43.406,158.337
C06944=1036.408,288.421,382.211,171.367,43.406,158.337
C06945=1036.414,288.668,382.180,171.371,43.408,158.338
C06946=1036.421,288.916,382.147,171.375,43.409,158.338
C06947=1036.427,289.164,382.116,171.379,43.410,158.339
C06948=1036.434,289.411,382.084,171.382,43.412,158.339
C06949=1036.442,289.660,382.052,171.386,43.412,158.340
C06950=1036.448,289.907,382.019,171.389,43.414,158.340
C06951=1036.455,290.155,381.988,171.394,43.415,158.341
C06952=1036.462,290.403,381.955,171.398,43.416,158.342
C06953=1036.468,290.651,381.924,171.402,43.417,158.342
C06954=1036.475,290.899,381.891,171.405,43.419,158.343
C06955=1036.484,291.248,381.846,171.410,43.420,158.344
C06956=1036.495,291.596,381.801,171.416,43.422,158.344
C06957=1036.504,291.945,381.756,171.421,43.424,158.345
C06958=1036.514,292.293,381.710,171.427,43.425,158.346
C06959=1036.521,292.541,381.678,171.431,43.426,158.347
C06960=1036.527,292.789,381.646,171.434,43.428,158.347
C06961=1036.535,293.037,381.614,171.438,43.429,158.348
C06962=1036.542,293.284,381.582,171.443,43.430,158.348
C06963=1036.548,293.532,381.550,171.446,43.431,158.349
C06964=1036.555,293.780,381.517,171.450,43.433,158.350
C06965=1036.562,294.028,381.484,171.454,43.433,158.350
C06966=1036.569,294.275,381.452,171.457,43.435,158.351
C06967=1036.575,294.523,381.420,171.462,43.436,158.351
C06968=1036.582,294.771,381.388,171.466,43.437,158.352
C06969=1036.589,295.019,381.355,171.469,43.438,158.352
C06970=1036.596,295.266,381.323,171.473,43.440,158.353
C06971=1036.603,295.515,381.290,171.477,43.441,158.354
C06972=1036.609,295.762,381.257,171.481,43.443,158.354
C06973=1036.616,296.009,381.225,171.485,43.444,158.355
C06974=1036.622,296.257,381.192,171.489,43.445,158.356
C06975=1036.629,296.505,381.159,171.493,43.446,158.356
C06976=1036.636,296.753,381.127,171.497,43.448,158.357
C06977=1036.642,297.000,381.094,171.500,43.450,158.357
C06978=1036.649,297.249,381.061,171.505,43.451,158.358
C06979=1036.656,297.496,381.028,171.509,43.452,158.359
C06980=1036.663,297.743,380.996,171.513,43.453,158.359
C06981=1036.670,297.992,380.963,171.516,43.455,158.360
C06982=1036.676,298.239,380.930,171.521,43.456,158.361
C06983=1036.683,298.488,380.897,171.525,43.457,158.361
C06984=1036.690,298.734,380.864,171.529,43.459,158.362
C06985=1036.696,298.982,380.831,171.532,43.460,158.362
C06986=1036.703,299.230,380.798,171.536,43.462,158.363
C06987=1036.710,299.478,380.766,171.541,43.463,158.364
C06988=1036.717,299.726,380.733,171.545,43.464,158.364
C06989=1036.723,299.973,380.700,171.548,43.466,158.365
C06990=1036.731,300.221,380.666,171.553,43.467,158.366
C06991=1036.737,300.469,380.634,171.557,43.469,158.366
C06992=1036.744,300.716,380.602,171.561,43.470,158.367
C06993=1036.751,300.964,380.568,171.565,43.472,158.368
C06994=1036.757,301.211,380.535,171.569,43.473,158.368
C06995=1036.764,301.459,380.502,171.573,43.474,158.369
C06996=1036.771,301.707,380.469,171.577,43.475,158.369
C06997=1036.779,301.954,380.436,171.582,43.477,158.370
C06998=1036.785,302.202,380.403,171.585,43.478,158.371
C06999=1036.792,302.450,380.370,171.589,43.480,158.371
C07000=1036.798,302.697,380.337,171.593,43.481,158.372
C07001=1036.806,302.945,380.304,171.598,43.483,158.373
C07002=1036.813,303.193,380.270,171.602,43.484,158.374
C07003=1036.820,303.440,380.238,171.605,43.486,158.374
C07004=1036.826,303.689,380.204,171.610,43.487,158.375
C07005=1036.833,303.936,380.171,171.614,43.489,158.376
C07006=1036.841,304.184,380.138,171.618,43.490,158.376
C07007=1036.847,304.431,380.105,171.622,43.491,158.377
C07008=1036.854,304.679,380.072,171.626,43.493,158.378
C07009=1036.861,304.927,380.038,171.630,43.494,158.378
C07010=1036.868,305.174,380.005,171.635,43.496,158.379
C07011=1036.879,305.539,379.957,171.641,43.498,158.380
C07012=1036.889,305.905,379.908,171.647,43.500,158.381
C07013=1036.899,306.270,379.858,171.653,43.502,158.382
C07014=1036.909,306.636,379.809,171.660,43.504,158.383
C07015=1036.917,306.883,379.776,171.663,43.506,158.383
C07016=1036.924,307.131,379.742,171.668,43.507,158.384
C07017=1036.930,307.379,379.709,171.672,43.509,158.385
C07018=1036.937,307.626,379.675,171.676,43.510,158.386
C07019=1036.945,307.874,379.642,171.680,43.512,158.386
C07020=1036.952,308.122,379.609,171.684,43.513,158.387
C07021=1036.959,308.369,379.575,171.689,43.514,158.388
C07022=1036.966,308.617,379.542,171.693,43.516,158.388
C07023=1036.973,308.864,379.508,171.698,43.517,158.389
C07024=1036.981,309.112,379.475,171.702,43.519,158.390
C07025=1036.987,309.359,379.442,171.706,43.521,158.390
C07026=1036.995,309.607,379.408,171.710,43.522,158.391
C07027=1037.002,309.855,379.374,171.714,43.524,158.392
C07028=1037.009,310.102,379.340,171.719,43.525,158.392
C07029=1037.016,310.350,379.307,171.723,43.527,158.393
C07030=1037.024,310.598,379.274,171.728,43.528,158.394
C07031=1037.030,310.845,379.241,171.732,43.530,158.395
C07032=1037.038,311.092,379.207,171.736,43.532,158.395
C07033=1037.045,311.340,379.173,171.740,43.533,158.396
C07034=1037.052,311.588,379.139,171.745,43.535,158.397
C07035=1037.059,311.836,379.105,171.749,43.536,158.397
C07036=1037.066,312.083,379.071,171.754,43.538,158.398
C07037=1037.072,312.330,379.037,171.758,43.539,158.399
C07038=1037.080,312.578,379.004,171.763,43.541,158.400
C07039=1037.087,312.826,378.970,171.767,43.543,158.400
C07040=1037.093,313.073,378.935,171.770,43.545,158.401
C07041=1037.100,313.320,378.901,171.775,43.547,158.402
C07042=1037.107,313.568,378.867,171.779,43.548,158.403
C07043=1037.114,313.816,378.833,171.784,43.550,158.403
C07044=1037.121,314.063,378.798,171.788,43.552,158.404
C07045=1037.128,314.311,378.764,171.793,43.554,158.405
C07046=1037.135,314.559,378.730,171.797,43.555,158.406
C07047=1037.141,314.806,378.696,171.802,43.557,158.406
C07048=1037.148,315.053,378.662,171.806,43.558,158.407
C07049=1037.155,315.301,378.627,171.811,43.560,158.408
C07050=1037.162,315.549,378.593,171.815,43.562,158.409
C07051=1037.169,315.796,378.559,171.820,43.564,158.410
C07052=1037.176,316.044,378.524,171.824,43.566,158.410
C07053=1037.183,316.291,378.490,171.828,43.567,158.411
C07054=1037.190,316.539,378.455,171.832,43.569,158.412
C07055=1037.197,316.786,378.422,171.837,43.571,158.413
C07056=1037.204,317.034,378.386,171.841,43.573,158.414
C07057=1037.211,317.281,378.353,171.846,43.575,158.414
C07058=1037.218,317.529,378.317,171.850,43.577,158.415
C07059=1037.225,317.776,378.284,171.855,43.578,158.416
C07060=1037.232,318.024,378.248,171.859,43.580,158.417
C07061=1037.239,318.271,378.215,171.864,43.582,158.417
C07062=1037.246,318.518,378.180,171.868,43.584,158.418
C07063=1037.253,318.766,378.146,171.873,43.585,158.419
C07064=1037.260,319.013,378.111,171.878,43.587,158.420
C07065=1037.267,319.261,378.076,171.882,43.589,158.420
C07066=1037.274,319.509,378.042,171.887,43.591,158.421
C07067=1037.285,319.879,377.990,171.894,43.594,158.423
C07068=1037.296,320.249,377.938,171.900,43.597,158.424
C07069=1037.306,320.619,377.887,171.907,43.599,158.425
C07070=1037.316,320.989,377.835,171.914,43.602,158.426
C07071=1037.324,321.237,377.800,171.919,43.604,158.427
C07072=1037.331,321.484,377.765,171.923,43.606,158.428
C07073=1037.338,321.732,377.731,171.928,43.608,158.429
C07074=1037.345,321.979,377.696,171.933,43.609,158.429
C07075=1037.353,322.227,377.661,171.937,43.612,158.430
C07076=1037.359,322.474,377.626,171.942,43.613,158.431
C07077=1037.367,322.722,377.591,171.947,43.615,158.432
C07078=1037.374,322.970,377.557,171.951,43.617,158.433
C07079=1037.381,323.217,377.522,171.956,43.619,158.434
C07080=1037.388,323.464,377.487,171.961,43.621,158.434
C07081=1037.396,323.712,377.452,171.965,43.623,158.435
C07082=1037.403,323.959,377.417,171.970,43.625,158.436
C07083=1037.411,324.206,377.383,171.975,43.627,158.437
C07084=1037.417,324.454,377.347,171.979,43.628,158.438
C07085=1037.425,324.701,377.313,171.984,43.631,158.439
C07086=1037.432,324.949,377.277,171.989,43.632,158.439
C07087=1037.440,325.196,377.243,171.993,43.634,158.440
C07088=1037.447,325.444,377.207,171.998,43.636,158.441
C07089=1037.455,325.691,377.173,172.003,43.638,158.442
C07090=1037.461,325.938,377.138,172.008,43.640,158.443
C07091=1037.469,326.186,377.103,172.012,43.642,158.444
C07092=1037.476,326.433,377.068,172.017,43.644,158.444
C07093=1037.484,326.680,377.033,172.022,43.646,158.445
C07094=1037.491,326.928,376.998,172.027,43.648,158.446
C07095=1037.498,327.176,376.962,172.031,43.650,158.447
C07096=1037.506,327.424,376.928,172.036,43.652,158.448
C07097=1037.513,327.670,376.892,172.042,43.654,158.449
C07098=1037.521,327.917,376.857,172.046,43.656,158.450
C07099=1037.528,328.165,376.822,172.051,43.658,158.451
C07100=1037.535,328.413,376.787,172.056,43.660,158.451
C07101=1037.543,328.661,376.752,172.061,43.662,158.452
C07102=1037.550,328.907,376.716,172.066,43.664,158.453
C07103=1037.557,329.155,376.680,172.070,43.666,158.454
C07104=1037.564,329.402,376.644,172.075,43.668,158.455
C07105=1037.571,329.649,376.609,172.080,43.671,158.456
C07106=1037.578,329.898,376.574,172.085,43.672,158.457
C07107=1037.586,330.144,376.538,172.089,43.675,158.458
C07108=1037.593,330.392,376.502,172.095,43.677,158.459
C07109=1037.600,330.639,376.467,172.100,43.679,158.460
C07110=1037.607,330.887,376.431,172.105,43.681,158.460
C07111=1037.615,331.134,376.396,172.109,43.683,158.461
C07112=1037.623,331.381,376.360,172.114,43.686,158.462
C07113=1037.630,331.628,376.325,172.119,43.688,158.463
C07114=1037.637,331.876,376.288,172.124,43.690,158.464
C07115=1037.644,332.123,376.253,172.130,43.692,158.465
C07116=1037.652,332.371,376.217,172.134,43.694,158.466
C07117=1037.659,332.617,376.181,172.139,43.696,158.467
C07118=1037.666,332.865,376.146,172.144,43.699,158.468
C07119=1037.673,333.112,376.110,172.149,43.701,158.469
C07120=1037.681,333.360,376.074,172.154,43.703,158.470
C07121=1037.688,333.607,376.038,172.159,43.705,158.471
C07122=1037.695,333.854,376.002,172.164,43.708,158.472
C07123=1037.706,334.220,375.949,172.171,43.711,158.473
C07124=1037.717,334.585,375.896,172.179,43.714,158.474
C07125=1037.728,334.951,375.843,172.187,43.717,158.476
C07126=1037.739,335.317,375.789,172.194,43.721,158.477
C07127=1037.746,335.564,375.754,172.199,43.723,158.478
C07128=1037.753,335.811,375.717,172.204,43.726,158.479
C07129=1037.761,336.059,375.681,172.209,43.728,158.480
C07130=1037.768,336.306,375.645,172.215,43.730,158.481
C07131=1037.775,336.553,375.608,172.220,43.732,158.482
C07132=1037.782,336.801,375.572,172.225,43.735,158.483
C07133=1037.789,337.047,375.536,172.230,43.737,158.484
C07134=1037.797,337.295,375.500,172.235,43.740,158.485
C07135=1037.805,337.542,375.463,172.240,43.742,158.486
C07136=1037.812,337.790,375.427,172.245,43.744,158.487
C07137=1037.819,338.037,375.391,172.250,43.747,158.488
C07138=1037.827,338.284,375.354,172.255,43.749,158.489
C07139=1037.834,338.531,375.318,172.261,43.752,158.490
C07140=1037.842,338.779,375.281,172.266,43.754,158.491
C07141=1037.849,339.026,375.245,172.271,43.756,158.492
C07142=1037.856,339.273,375.209,172.276,43.759,158.493
C07143=1037.864,339.520,375.172,172.282,43.761,158.494
C07144=1037.872,339.767,375.136,172.287,43.763,158.495
C07145=1037.879,340.015,375.099,172.292,43.766,158.496
C07146=1037.886,340.261,375.062,172.297,43.768,158.497
C07147=1037.894,340.509,375.026,172.303,43.771,158.498
C07148=1037.902,340.756,374.990,172.308,43.773,158.499
C07149=1037.909,341.003,374.952,172.313,43.776,158.500
C07150=1037.916,341.251,374.916,172.319,43.778,158.501
C07151=1037.924,341.498,374.880,172.324,43.781,158.502
C07152=1037.931,341.745,374.842,172.329,43.783,158.503
C07153=1037.939,341.993,374.806,172.335,43.786,158.504
C07154=1037.946,342.239,374.769,172.340,43.788,158.505
C07155=1037.953,342.487,374.733,172.345,43.791,158.506
C07156=1037.961,342.734,374.695,172.351,43.794,158.508
C07157=1037.969,342.981,374.658,172.356,43.796,158.509
C07158=1037.975,343.228,374.621,172.361,43.799,158.510
C07159=1037.983,343.475,374.584,172.366,43.801,158.511
C07160=1037.990,343.723,374.548,172.372,43.804,158.512
C07161=1037.998,343.970,374.511,172.377,43.806,158.513
C07162=1038.006,344.217,374.473,172.382,43.809,158.514
C07163=1038.014,344.464,374.436,172.388,43.811,158.515
C07164=1038.021,344.711,374.399,172.393,43.814,158.516
C07165=1038.029,344.958,374.363,172.399,43.816,158.517
C07166=1038.036,345.205,374.325,172.404,43.819,158.518
C07167=1038.044,345.452,374.288,172.409,43.822,158.519
C07168=1038.051,345.700,374.251,172.415,43.825,158.521
C07169=1038.058,345.947,374.214,172.421,43.827,158.522
C07170=1038.066,346.194,374.177,172.427,43.830,158.523
C07171=1038.073,346.441,374.139,172.432,43.832,158.524
C07172=1038.081,346.688,374.102,172.437,43.835,158.525
C07173=1038.088,346.935,374.065,172.443,43.838,158.526
C07174=1038.096,347.182,374.027,172.448,43.841,158.527
C07175=1038.104,347.429,373.990,172.454,43.844,158.528
C07176=1038.111,347.676,373.953,172.459,43.846,158.529
C07177=1038.119,347.924,373.915,172.465,43.848,158.530
C07178=1038.127,348.171,373.878,172.471,43.851,158.532
C07179=1038.137,348.533,373.823,172.479,43.855,158.533
C07180=1038.149,348.895,373.768,172.487,43.859,158.535
C07181=1038.160,349.256,373.713,172.495,43.864,158.537
C07182=1038.171,349.619,373.658,172.503,43.867,158.538
C07183=1038.178,349.866,373.621,172.509,43.871,158.540
C07184=1038.186,350.113,373.583,172.515,43.873,158.541
C07185=1038.194,350.360,373.546,172.521,43.876,158.542
C07186=1038.202,350.607,373.508,172.526,43.879,158.543
C07187=1038.209,350.854,373.470,172.532,43.882,158.544
C07188=1038.217,351.101,373.432,172.537,43.884,158.545
C07189=1038.224,351.348,373.395,172.544,43.887,158.547
C07190=1038.232,351.595,373.356,172.549,43.890,158.548
C07191=1038.240,351.842,373.319,172.555,43.893,158.549
C07192=1038.248,352.089,373.281,172.560,43.896,158.550
C07193=1038.255,352.337,373.243,172.566,43.899,158.551
C07194=1038.263,352.583,373.205,172.572,43.902,158.552
C07195=1038.270,352.830,373.167,172.578,43.905,158.554
C07196=1038.278,353.077,373.129,172.583,43.908,158.555
C07197=1038.286,353.325,373.091,172.589,43.911,158.556
C07198=1038.293,353.571,373.053,172.595,43.913,158.557
C07199=1038.302,353.818,373.015,172.601,43.917,158.559
C07200=1038.309,354.065,372.977,172.606,43.919,158.560
C07201=1038.317,354.312,372.939,172.613,43.923,158.561
C07202=1038.325,354.559,372.901,172.619,43.925,158.562
C07203=1038.332,354.806,372.863,172.624,43.928,158.563
C07204=1038.340,355.053,372.824,172.631,43.931,158.565
C07205=1038.348,355.300,372.786,172.636,43.934,158.566
C07206=1038.355,355.547,372.748,172.642,43.937,158.567
C07207=1038.363,355.794,372.710,172.648,43.940,158.568
C07208=1038.371,356.041,372.672,172.654,43.943,158.570
C07209=1038.380,356.287,372.634,172.660,43.947,158.571
C07210=1038.387,356.534,372.595,172.666,43.949,158.572
C07211=1038.395,356.782,372.556,172.672,43.953,158.573
C07212=1038.402,357.028,372.518,172.677,43.955,158.575
C07213=1038.410,357.275,372.479,172.684,43.958,158.576
C07214=1038.418,357.522,372.441,172.690,43.962,158.577
C07215=1038.426,357.769,372.402,172.695,43.965,158.578
C07216=1038.434,358.016,372.364,172.702,43.968,158.580
C07217=1038.442,358.263,372.326,172.708,43.971,158.581
C07218=1038.450,358.510,372.287,172.714,43.974,158.582
C07219=1038.458,358.756,372.249,172.720,43.978,158.584
C07220=1038.466,359.004,372.210,172.727,43.981,158.585
C07221=1038.472,359.251,372.171,172.732,43.983,158.586
C07222=1038.481,359.498,372.133,172.738,43.987,158.587
C07223=1038.489,359.744,372.093,172.744,43.990,158.589
C07224=1038.497,359.991,372.055,172.750,43.993,158.590
C07225=1038.505,360.238,372.016,172.757,43.996,158.591
C07226=1038.513,360.485,371.978,172.763,44.000,158.593
C07227=1038.521,360.731,371.939,172.769,44.003,158.594
C07228=1038.528,360.979,371.900,172.775,44.006,158.595
C07229=1038.536,361.226,371.861,172.782,44.009,158.597
C07230=1038.544,361.472,371.822,172.787,44.013,158.598
C07231=1038.552,361.719,371.784,172.794,44.016,158.599
C07232=1038.561,361.966,371.744,172.800,44.019,158.601
C07233=1038.568,362.212,371.705,172.807,44.022,158.602
C07234=1038.576,362.459,371.666,172.812,44.026,158.603
C07235=1038.588,362.828,371.607,172.822,44.031,158.605
C07236=1038.599,363.195,371.549,172.832,44.036,158.608
C07237=1038.612,363.564,371.491,172.840,44.041,158.610
C07238=1038.623,363.932,371.432,172.850,44.046,158.612
C07239=1038.631,364.179,371.393,172.857,44.049,158.613
C07240=1038.639,364.425,371.354,172.862,44.052,158.614
C07241=1038.647,364.672,371.314,172.869,44.056,158.616
C07242=1038.655,364.918,371.275,172.875,44.059,158.617
C07243=1038.663,365.165,371.235,172.882,44.063,158.619
C07244=1038.671,365.412,371.196,172.888,44.067,158.620
C07245=1038.678,365.659,371.156,172.894,44.070,158.621
C07246=1038.687,365.906,371.117,172.901,44.073,158.623
C07247=1038.695,366.153,371.077,172.907,44.077,158.624
C07248=1038.703,366.399,371.038,172.914,44.080,158.626
C07249=1038.712,366.646,370.998,172.921,44.083,158.627
C07250=1038.719,366.893,370.959,172.927,44.087,158.629
C07251=1038.728,367.139,370.919,172.934,44.091,158.630
C07252=1038.735,367.386,370.879,172.940,44.094,158.632
C07253=1038.744,367.633,370.840,172.946,44.098,158.633
C07254=1038.752,367.880,370.800,172.953,44.101,158.634
C07255=1038.760,368.126,370.761,172.960,44.105,158.636
C07256=1038.768,368.373,370.720,172.966,44.109,158.637
C07257=1038.777,368.619,370.681,172.973,44.112,158.639
C07258=1038.784,368.866,370.641,172.980,44.115,158.640
C07259=1038.793,369.113,370.601,172.986,44.119,158.642
C07260=1038.800,369.360,370.562,172.993,44.123,158.643
C07261=1038.809,369.606,370.522,172.999,44.126,158.645
C07262=1038.818,369.852,370.482,173.006,44.130,158.646
C07263=1038.825,370.099,370.442,173.012,44.134,158.648
C07264=1038.833,370.345,370.402,173.019,44.137,158.649
C07265=1038.842,370.593,370.362,173.026,44.141,158.651
C07266=1038.850,370.840,370.322,173.033,44.145,158.652
C07267=1038.858,371.086,370.281,173.039,44.149,158.654
C07268=1038.866,371.332,370.241,173.046,44.152,158.655
C07269=1038.875,371.579,370.201,173.053,44.156,158.657
C07270=1038.883,371.825,370.161,173.060,44.159,158.658
C07271=1038.890,372.072,370.121,173.066,44.163,158.660
C07272=1038.899,372.319,370.080,173.073,44.168,158.662
C07273=1038.907,372.565,370.039,173.080,44.171,158.663
C07274=1038.916,372.812,370.000,173.087,44.175,158.665
C07275=1038.924,373.058,369.959,173.094,44.179,158.666
C07276=1038.932,373.304,369.919,173.100,44.182,158.668
C07277=1038.940,373.551,369.878,173.108,44.187,158.669
C07278=1038.948,373.798,369.838,173.115,44.190,158.671
C07279=1038.957,374.044,369.798,173.121,44.194,158.672
C07280=1038.965,374.291,369.757,173.128,44.198,158.674
C07281=1038.973,374.538,369.716,173.136,44.202,158.676
C07282=1038.981,374.784,369.675,173.143,44.206,158.677
C07283=1038.990,375.031,369.634,173.150,44.210,158.679
